LIN {X 0,Y 471.036,Z 185.812,A -85,B 0,C 180,E1 -7424.234,E2 -7424.234} C_VEL
LIN {X 0,Y 468.624,Z 186.111,A -85,B 0,C 180,E1 -7425.161,E2 -7425.161} C_VEL
LIN {X 0,Y 467.615,Z 186.239,A -85,B 0,C 180,E1 -7425.877,E2 -7425.877} C_VEL
LIN {X 0,Y 467.546,Z 186.246,A -85,B 0,C 180,E1 -7426.119,E2 -7426.119} C_VEL
LIN {X 0,Y 467.577,Z 186.237,A -85,B 0,C 180,E1 -7428.723,E2 -7428.723} C_VEL
LIN {X 0,Y 467.564,Z 186.243,A -85,B 0,C 180,E1 -7431.955,E2 -7431.955} C_VEL
LIN {X 0,Y 467.566,Z 186.241,A -85,B 0,C 180,E1 -7435.167,E2 -7435.167} C_VEL
LIN {X 0,Y 467.581,Z 186.237,A -85,B 0,C 180,E1 -7438.259,E2 -7438.259} C_VEL
LIN {X 0,Y 467.576,Z 186.241,A -85,B 0,C 180,E1 -7441.25,E2 -7441.25} C_VEL
LIN {X 0,Y 467.611,Z 186.234,A -85,B 0,C 180,E1 -7444.16,E2 -7444.16} C_VEL
LIN {X 0,Y 467.575,Z 186.24,A -85,B 0,C 180,E1 -7446.995,E2 -7446.995} C_VEL
LIN {X 0,Y 467.621,Z 186.235,A -85,B 0,C 180,E1 -7449.777,E2 -7449.777} C_VEL
LIN {X 0,Y 467.605,Z 186.234,A -85,B 0,C 180,E1 -7452.506,E2 -7452.506} C_VEL
LIN {X 0,Y 467.608,Z 186.24,A -85,B 0,C 180,E1 -7455.196,E2 -7455.196} C_VEL
LIN {X 0,Y 467.654,Z 186.229,A -85,B 0,C 180,E1 -7457.854,E2 -7457.854} C_VEL
LIN {X 0,Y 467.68,Z 186.23,A -85,B 0,C 180,E1 -7461.357,E2 -7461.357} C_VEL
LIN {X 0,Y 467.743,Z 186.217,A -85,B 0,C 180,E1 -7463.962,E2 -7463.962} C_VEL
LIN {X 0,Y 467.857,Z 186.206,A -85,B 0,C 180,E1 -7467.417,E2 -7467.417} C_VEL
LIN {X 0,Y 467.88,Z 186.199,A -85,B 0,C 180,E1 -7469.999,E2 -7469.999} C_VEL
LIN {X 0,Y 467.857,Z 186.204,A -85,B 0,C 180,E1 -7472.582,E2 -7472.582} C_VEL
LIN {X 0,Y 467.732,Z 186.218,A -85,B 0,C 180,E1 -7476.037,E2 -7476.037} C_VEL
LIN {X 0,Y 467.678,Z 186.228,A -85,B 0,C 180,E1 -7478.642,E2 -7478.642} C_VEL
LIN {X 0,Y 467.652,Z 186.228,A -85,B 0,C 180,E1 -7482.145,E2 -7482.145} C_VEL
LIN {X 0,Y 467.635,Z 186.23,A -85,B 0,C 180,E1 -7485.694,E2 -7485.694} C_VEL
LIN {X 0,Y 467.613,Z 186.241,A -85,B 0,C 180,E1 -7488.764,E2 -7488.764} C_VEL
LIN {X 0,Y 467.576,Z 186.239,A -85,B 0,C 180,E1 -7491.268,E2 -7491.268} C_VEL
LIN {X 0,Y 467.568,Z 186.238,A -85,B 0,C 180,E1 -7493.943,E2 -7493.943} C_VEL
LIN {X 0,Y 467.623,Z 186.238,A -85,B 0,C 180,E1 -7496.799,E2 -7496.799} C_VEL
LIN {X 0,Y 467.548,Z 186.241,A -85,B 0,C 180,E1 -7499.737,E2 -7499.737} C_VEL
LIN {X 0,Y 467.577,Z 186.243,A -85,B 0,C 180,E1 -7502.758,E2 -7502.758} C_VEL
LIN {X 0,Y 467.55,Z 186.241,A -85,B 0,C 180,E1 -7505.889,E2 -7505.889} C_VEL
LIN {X 0,Y 467.592,Z 186.236,A -85,B 0,C 180,E1 -7509.142,E2 -7509.142} C_VEL
LIN {X 0,Y 467.611,Z 186.239,A -85,B 0,C 180,E1 -7512.571,E2 -7512.571} C_VEL
LIN {X 0,Y 467.562,Z 186.24,A -85,B 0,C 180,E1 -7515.053,E2 -7515.053} C_VEL
LIN {X 0,Y 467.58,Z 186.237,A -85,B 0,C 180,E1 -7517.44,E2 -7517.44} C_VEL
LIN {X 0,Y 467.591,Z 186.237,A -85,B 0,C 180,E1 -7520.857,E2 -7520.857} C_VEL
LIN {X 0,Y 467.555,Z 186.248,A -85,B 0,C 180,E1 -7524.26,E2 -7524.26} C_VEL
LIN {X 0,Y 467.574,Z 186.237,A -85,B 0,C 180,E1 -7527.321,E2 -7527.321} C_VEL
LIN {X 0,Y 467.569,Z 186.24,A -85,B 0,C 180,E1 -7530.665,E2 -7530.665} C_VEL
LIN {X 0,Y 467.607,Z 186.233,A -85,B 0,C 180,E1 -7533.2,E2 -7533.2} C_VEL
LIN {X 0,Y 467.584,Z 186.239,A -85,B 0,C 180,E1 -7536.468,E2 -7536.468} C_VEL
LIN {X 0,Y 467.615,Z 186.237,A -85,B 0,C 180,E1 -7539.777,E2 -7539.777} C_VEL
LIN {X 0,Y 467.6,Z 186.236,A -85,B 0,C 180,E1 -7542.507,E2 -7542.507} C_VEL
LIN {X 0,Y 467.597,Z 186.235,A -85,B 0,C 180,E1 -7545.197,E2 -7545.197} C_VEL
LIN {X 0,Y 467.648,Z 186.236,A -85,B 0,C 180,E1 -7547.855,E2 -7547.855} C_VEL
LIN {X 0,Y 467.673,Z 186.227,A -85,B 0,C 180,E1 -7551.358,E2 -7551.358} C_VEL
LIN {X 0,Y 467.734,Z 186.223,A -85,B 0,C 180,E1 -7553.963,E2 -7553.963} C_VEL
LIN {X 0,Y 467.85,Z 186.207,A -85,B 0,C 180,E1 -7557.417,E2 -7557.417} C_VEL
LIN {X 0,Y 467.873,Z 186.204,A -85,B 0,C 180,E1 -7560,E2 -7560} C_VEL
LIN {X 0,Y 467.851,Z 186.203,A -85,B 0,C 180,E1 -7562.583,E2 -7562.583} C_VEL
LIN {X 0,Y 467.726,Z 186.221,A -85,B 0,C 180,E1 -7566.038,E2 -7566.038} C_VEL
LIN {X 0,Y 467.672,Z 186.225,A -85,B 0,C 180,E1 -7568.643,E2 -7568.643} C_VEL
LIN {X 0,Y 467.648,Z 186.229,A -85,B 0,C 180,E1 -7572.146,E2 -7572.146} C_VEL
LIN {X 0,Y 467.631,Z 186.235,A -85,B 0,C 180,E1 -7575.696,E2 -7575.696} C_VEL
LIN {X 0,Y 467.61,Z 186.234,A -85,B 0,C 180,E1 -7578.765,E2 -7578.765} C_VEL
LIN {X 0,Y 467.573,Z 186.245,A -85,B 0,C 180,E1 -7581.269,E2 -7581.269} C_VEL
LIN {X 0,Y 467.563,Z 186.24,A -85,B 0,C 180,E1 -7583.944,E2 -7583.944} C_VEL
LIN {X 0,Y 467.609,Z 186.235,A -85,B 0,C 180,E1 -7586.801,E2 -7586.801} C_VEL
LIN {X 0,Y 467.547,Z 186.242,A -85,B 0,C 180,E1 -7589.739,E2 -7589.739} C_VEL
LIN {X 0,Y 467.573,Z 186.24,A -85,B 0,C 180,E1 -7592.76,E2 -7592.76} C_VEL
LIN {X 0,Y 467.547,Z 186.241,A -85,B 0,C 180,E1 -7595.891,E2 -7595.891} C_VEL
LIN {X 0,Y 467.571,Z 186.245,A -85,B 0,C 180,E1 -7599.146,E2 -7599.146} C_VEL
LIN {X 0,Y 467.583,Z 186.239,A -85,B 0,C 180,E1 -7602.568,E2 -7602.568} C_VEL
LIN {X 0,Y 467.567,Z 186.245,A -85,B 0,C 180,E1 -7605.054,E2 -7605.054} C_VEL
LIN {X 0,Y 467.569,Z 186.242,A -85,B 0,C 180,E1 -7608.598,E2 -7608.598} C_VEL
LIN {X 0,Y 467.559,Z 186.239,A -85,B 0,C 180,E1 -7611.956,E2 -7611.956} C_VEL
LIN {X 0,Y 467.561,Z 186.245,A -85,B 0,C 180,E1 -7615.168,E2 -7615.168} C_VEL
LIN {X 0,Y 467.581,Z 186.242,A -85,B 0,C 180,E1 -7618.261,E2 -7618.261} C_VEL
LIN {X 0,Y 467.555,Z 186.247,A -85,B 0,C 180,E1 -7621.25,E2 -7621.25} C_VEL
LIN {X 0,Y 467.616,Z 186.484,A -85,B 0,C 180,E1 -7622.478,E2 -7622.478} C_VEL
LIN {X 0,Y 471.107,Z 202.041,A -85,B 0,C 180,E1 -7624.84,E2 -7624.84} C_VEL
LIN {X 0,Y 470.606,Z 215.622,A -85,B 0,C 180,E1 -7626.688,E2 -7626.688} C_VEL
LIN {X 0,Y 469.516,Z 239.357,A -85,B 0,C 180,E1 -7629.863,E2 -7629.863} C_VEL
LIN {X 0,Y 468.66,Z 261.512,A -85,B 0,C 180,E1 -7632.796,E2 -7632.796} C_VEL
LIN {X 0,Y 468.555,Z 265.454,A -85,B 0,C 180,E1 -7633.297,E2 -7633.297} C_VEL
LIN {X 0,Y 470.521,Z 284.051,A -85,B 0,C 180,E1 -7633.671,E2 -7633.671} C_VEL
LIN {X 0,Y 469.828,Z 373.176,A -85,B 0,C 180,E1 -7635.103,E2 -7635.103} C_VEL
LIN {X 0,Y 469.492,Z 386.416,A -85,B 0,C 180,E1 -7635.48,E2 -7635.48} C_VEL
LIN {X 0,Y 469.075,Z 399.132,A -85,B 0,C 180,E1 -7636.02,E2 -7636.02} C_VEL
LIN {X 0,Y 468.644,Z 410.397,A -85,B 0,C 180,E1 -7636.67,E2 -7636.67} C_VEL
LIN {X 0,Y 468.245,Z 421.339,A -85,B 0,C 180,E1 -7637.479,E2 -7637.479} C_VEL
LIN {X 0,Y 467.741,Z 432.571,A -85,B 0,C 180,E1 -7638.517,E2 -7638.517} C_VEL
LIN {X 0,Y 467.393,Z 441.968,A -85,B 0,C 180,E1 -7639.605,E2 -7639.605} C_VEL
LIN {X 0,Y 467.101,Z 451.067,A -85,B 0,C 180,E1 -7640.911,E2 -7640.911} C_VEL
LIN {X 0,Y 466.93,Z 458.368,A -85,B 0,C 180,E1 -7642.215,E2 -7642.215} C_VEL
LIN {X 0,Y 466.842,Z 464.127,A -85,B 0,C 180,E1 -7643.51,E2 -7643.51} C_VEL
LIN {X 0,Y 466.787,Z 468.686,A -85,B 0,C 180,E1 -7644.818,E2 -7644.818} C_VEL
LIN {X 0,Y 466.785,Z 471.065,A -85,B 0,C 180,E1 -7645.683,E2 -7645.683} C_VEL
LIN {X 0,Y 466.872,Z 473.007,A -85,B 0,C 180,E1 -7646.549,E2 -7646.549} C_VEL
LIN {X 0,Y 466.84,Z 474.474,A -85,B 0,C 180,E1 -7647.412,E2 -7647.412} C_VEL
LIN {X 0,Y 466.727,Z 476.099,A -85,B 0,C 180,E1 -7649.138,E2 -7649.138} C_VEL
LIN {X 0,Y 466.746,Z 476.31,A -85,B 0,C 180,E1 -7650.001,E2 -7650.001} C_VEL
LIN {X 0,Y 466.73,Z 476.064,A -85,B 0,C 180,E1 -7650.863,E2 -7650.863} C_VEL
LIN {X 0,Y 466.843,Z 474.348,A -85,B 0,C 180,E1 -7652.589,E2 -7652.589} C_VEL
LIN {X 0,Y 466.886,Z 472.858,A -85,B 0,C 180,E1 -7653.453,E2 -7653.453} C_VEL
LIN {X 0,Y 466.748,Z 469.736,A -85,B 0,C 180,E1 -7654.751,E2 -7654.751} C_VEL
LIN {X 0,Y 466.788,Z 465.534,A -85,B 0,C 180,E1 -7656.05,E2 -7656.05} C_VEL
LIN {X 0,Y 466.931,Z 460.123,A -85,B 0,C 180,E1 -7657.351,E2 -7657.351} C_VEL
LIN {X 0,Y 467.007,Z 453.309,A -85,B 0,C 180,E1 -7658.656,E2 -7658.656} C_VEL
LIN {X 0,Y 467.237,Z 444.849,A -85,B 0,C 180,E1 -7659.962,E2 -7659.962} C_VEL
LIN {X 0,Y 467.616,Z 436.186,A -85,B 0,C 180,E1 -7661.048,E2 -7661.048} C_VEL
LIN {X 0,Y 467.936,Z 427.836,A -85,B 0,C 180,E1 -7661.919,E2 -7661.919} C_VEL
LIN {X 0,Y 468.328,Z 416.572,A -85,B 0,C 180,E1 -7662.876,E2 -7662.876} C_VEL
LIN {X 0,Y 468.788,Z 404.931,A -85,B 0,C 180,E1 -7663.658,E2 -7663.658} C_VEL
LIN {X 0,Y 469.334,Z 392.149,A -85,B 0,C 180,E1 -7664.305,E2 -7664.305} C_VEL
LIN {X 0,Y 469.711,Z 379.318,A -85,B 0,C 180,E1 -7664.764,E2 -7664.764} C_VEL
LIN {X 0,Y 469.972,Z 365.957,A -85,B 0,C 180,E1 -7665.06,E2 -7665.06} C_VEL
LIN {X 0,Y 470.591,Z 282.438,A -85,B 0,C 180,E1 -7666.414,E2 -7666.414} C_VEL
LIN {X 0,Y 468.55,Z 264.229,A -85,B 0,C 180,E1 -7666.822,E2 -7666.822} C_VEL
LIN {X 0,Y 469.271,Z 242.062,A -85,B 0,C 180,E1 -7669.647,E2 -7669.647} C_VEL
LIN {X 0,Y 470.196,Z 217.219,A -85,B 0,C 180,E1 -7672.869,E2 -7672.869} C_VEL
LIN {X 0,Y 470.821,Z 201.375,A -85,B 0,C 180,E1 -7674.942,E2 -7674.942} C_VEL
LIN {X 0,Y 468.587,Z 190.486,A -85,B 0,C 180,E1 -7676.531,E2 -7676.531} C_VEL
LIN {X 0,Y 467.615,Z 186.372,A -85,B 0,C 180,E1 -7677.184,E2 -7677.184} C_VEL
LIN {X 0,Y 467.569,Z 186.245,A -85,B 0,C 180,E1 -7680.734,E2 -7680.734} C_VEL
LIN {X 0,Y 467.573,Z 186.243,A -85,B 0,C 180,E1 -7683.79,E2 -7683.79} C_VEL
LIN {X 0,Y 467.527,Z 186.25,A -85,B 0,C 180,E1 -7686.963,E2 -7686.963} C_VEL
LIN {X 0,Y 467.567,Z 186.241,A -85,B 0,C 180,E1 -7689.952,E2 -7689.952} C_VEL
LIN {X 0,Y 467.545,Z 186.246,A -85,B 0,C 180,E1 -7692.565,E2 -7692.565} C_VEL
LIN {X 0,Y 467.568,Z 186.246,A -85,B 0,C 180,E1 -7695.052,E2 -7695.052} C_VEL
LIN {X 0,Y 467.575,Z 186.241,A -85,B 0,C 180,E1 -7698.596,E2 -7698.596} C_VEL
LIN {X 0,Y 467.567,Z 186.239,A -85,B 0,C 180,E1 -7701.955,E2 -7701.955} C_VEL
LIN {X 0,Y 467.561,Z 186.244,A -85,B 0,C 180,E1 -7705.167,E2 -7705.167} C_VEL
LIN {X 0,Y 467.584,Z 186.24,A -85,B 0,C 180,E1 -7708.26,E2 -7708.26} C_VEL
LIN {X 0,Y 467.577,Z 186.241,A -85,B 0,C 180,E1 -7711.25,E2 -7711.25} C_VEL
LIN {X 0,Y 467.599,Z 186.238,A -85,B 0,C 180,E1 -7714.159,E2 -7714.159} C_VEL
LIN {X 0,Y 467.578,Z 186.241,A -85,B 0,C 180,E1 -7716.995,E2 -7716.995} C_VEL
LIN {X 0,Y 467.623,Z 186.233,A -85,B 0,C 180,E1 -7719.777,E2 -7719.777} C_VEL
LIN {X 0,Y 467.597,Z 186.241,A -85,B 0,C 180,E1 -7722.506,E2 -7722.506} C_VEL
LIN {X 0,Y 467.606,Z 186.237,A -85,B 0,C 180,E1 -7725.196,E2 -7725.196} C_VEL
LIN {X 0,Y 467.657,Z 186.23,A -85,B 0,C 180,E1 -7727.854,E2 -7727.854} C_VEL
LIN {X 0,Y 467.671,Z 186.228,A -85,B 0,C 180,E1 -7731.357,E2 -7731.357} C_VEL
LIN {X 0,Y 467.721,Z 186.226,A -85,B 0,C 180,E1 -7733.962,E2 -7733.962} C_VEL
LIN {X 0,Y 467.859,Z 186.208,A -85,B 0,C 180,E1 -7737.417,E2 -7737.417} C_VEL
LIN {X 0,Y 467.821,Z 186.447,A -85,B 0,C 180,E1 -7739.112,E2 -7739.112} C_VEL
LIN {X 0,Y 468.474,Z 190.11,A -85,B 0,C 180,E1 -7739.785,E2 -7739.785} C_VEL
LIN {X 0,Y 468.367,Z 206.386,A -85,B 0,C 180,E1 -7742.58,E2 -7742.58} C_VEL
LIN {X 0,Y 468.286,Z 223.54,A -85,B 0,C 180,E1 -7745.598,E2 -7745.598} C_VEL
LIN {X 0,Y 468.274,Z 227.237,A -85,B 0,C 180,E1 -7746.219,E2 -7746.219} C_VEL
LIN {X 0,Y 470.377,Z 238.502,A -85,B 0,C 180,E1 -7746.541,E2 -7746.541} C_VEL
LIN {X 0,Y 469.573,Z 308.823,A -85,B 0,C 180,E1 -7747.834,E2 -7747.834} C_VEL
LIN {X 0,Y 469.438,Z 320.442,A -85,B 0,C 180,E1 -7748.211,E2 -7748.211} C_VEL
LIN {X 0,Y 469.166,Z 332.332,A -85,B 0,C 180,E1 -7748.791,E2 -7748.791} C_VEL
LIN {X 0,Y 468.847,Z 342.842,A -85,B 0,C 180,E1 -7749.49,E2 -7749.49} C_VEL
LIN {X 0,Y 468.516,Z 353.004,A -85,B 0,C 180,E1 -7750.37,E2 -7750.37} C_VEL
LIN {X 0,Y 468.196,Z 361.041,A -85,B 0,C 180,E1 -7751.252,E2 -7751.252} C_VEL
LIN {X 0,Y 467.882,Z 368.755,A -85,B 0,C 180,E1 -7752.303,E2 -7752.303} C_VEL
LIN {X 0,Y 467.622,Z 375.472,A -85,B 0,C 180,E1 -7753.471,E2 -7753.471} C_VEL
LIN {X 0,Y 467.334,Z 381.402,A -85,B 0,C 180,E1 -7754.812,E2 -7754.812} C_VEL
LIN {X 0,Y 467.168,Z 385.738,A -85,B 0,C 180,E1 -7756.159,E2 -7756.159} C_VEL
LIN {X 0,Y 466.985,Z 388.645,A -85,B 0,C 180,E1 -7757.517,E2 -7757.517} C_VEL
LIN {X 0,Y 466.938,Z 389.95,A -85,B 0,C 180,E1 -7758.517,E2 -7758.517} C_VEL
LIN {X 0,Y 466.891,Z 390.505,A -85,B 0,C 180,E1 -7759.339,E2 -7759.339} C_VEL
LIN {X 0,Y 466.89,Z 390.575,A -85,B 0,C 180,E1 -7760.255,E2 -7760.255} C_VEL
LIN {X 0,Y 466.896,Z 390.092,A -85,B 0,C 180,E1 -7761.177,E2 -7761.177} C_VEL
LIN {X 0,Y 466.919,Z 388.996,A -85,B 0,C 180,E1 -7762.104,E2 -7762.104} C_VEL
LIN {X 0,Y 467.041,Z 386.528,A -85,B 0,C 180,E1 -7763.376,E2 -7763.376} C_VEL
LIN {X 0,Y 467.169,Z 383.529,A -85,B 0,C 180,E1 -7764.437,E2 -7764.437} C_VEL
LIN {X 0,Y 467.36,Z 378.061,A -85,B 0,C 180,E1 -7765.854,E2 -7765.854} C_VEL
LIN {X 0,Y 467.522,Z 372.051,A -85,B 0,C 180,E1 -7767.026,E2 -7767.026} C_VEL
LIN {X 0,Y 467.789,Z 365.797,A -85,B 0,C 180,E1 -7768.001,E2 -7768.001} C_VEL
LIN {X 0,Y 468.081,Z 357.37,A -85,B 0,C 180,E1 -7769.057,E2 -7769.057} C_VEL
LIN {X 0,Y 468.372,Z 348.64,A -85,B 0,C 180,E1 -7769.928,E2 -7769.928} C_VEL
LIN {X 0,Y 468.723,Z 338.054,A -85,B 0,C 180,E1 -7770.754,E2 -7770.754} C_VEL
LIN {X 0,Y 468.99,Z 327.029,A -85,B 0,C 180,E1 -7771.405,E2 -7771.405} C_VEL
LIN {X 0,Y 469.178,Z 314.743,A -85,B 0,C 180,E1 -7771.919,E2 -7771.919} C_VEL
LIN {X 0,Y 469.307,Z 301.965,A -85,B 0,C 180,E1 -7772.241,E2 -7772.241} C_VEL
LIN {X 0,Y 469.804,Z 237.356,A -85,B 0,C 180,E1 -7773.338,E2 -7773.338} C_VEL
LIN {X 0,Y 467.979,Z 226.462,A -85,B 0,C 180,E1 -7773.612,E2 -7773.612} C_VEL
LIN {X 0,Y 468.255,Z 209.645,A -85,B 0,C 180,E1 -7776.895,E2 -7776.895} C_VEL
LIN {X 0,Y 468.539,Z 193.341,A -85,B 0,C 180,E1 -7780.164,E2 -7780.164} C_VEL
LIN {X 0,Y 468.184,Z 189.189,A -85,B 0,C 180,E1 -7781.023,E2 -7781.023} C_VEL
LIN {X 0,Y 467.629,Z 186.277,A -85,B 0,C 180,E1 -7781.702,E2 -7781.702} C_VEL
LIN {X 0,Y 467.564,Z 186.243,A -85,B 0,C 180,E1 -7785.052,E2 -7785.052} C_VEL
LIN {X 0,Y 467.546,Z 186.246,A -85,B 0,C 180,E1 -7786.119,E2 -7786.119} C_VEL
LIN {X 0,Y 466.92,Z 186.33,A -85,B 0,C 180,E1 -7786.838,E2 -7786.838} C_VEL
LIN {X 0,Y 464.09,Z 186.689,A -85,B 0,C 180,E1 -7788.007,E2 -7788.007} C_VEL
LIN {X 0,Y 461.667,Z 186.988,A -85,B 0,C 180,E1 -7788.949,E2 -7788.949} C_VEL
LIN {X 0,Y 460.617,Z 187.112,A -85,B 0,C 180,E1 -7789.677,E2 -7789.677} C_VEL
LIN {X 0,Y 460.528,Z 187.12,A -85,B 0,C 180,E1 -7789.924,E2 -7789.924} C_VEL
LIN {X 0,Y 460.499,Z 187.119,A -85,B 0,C 180,E1 -7792.523,E2 -7792.523} C_VEL
LIN {X 0,Y 460.547,Z 187.121,A -85,B 0,C 180,E1 -7795.623,E2 -7795.623} C_VEL
LIN {X 0,Y 460.535,Z 187.114,A -85,B 0,C 180,E1 -7798.744,E2 -7798.744} C_VEL
LIN {X 0,Y 460.587,Z 187.108,A -85,B 0,C 180,E1 -7802.252,E2 -7802.252} C_VEL
LIN {X 0,Y 460.558,Z 187.112,A -85,B 0,C 180,E1 -7804.705,E2 -7804.705} C_VEL
LIN {X 0,Y 460.509,Z 187.124,A -85,B 0,C 180,E1 -7807.571,E2 -7807.571} C_VEL
LIN {X 0,Y 460.567,Z 187.11,A -85,B 0,C 180,E1 -7810.384,E2 -7810.384} C_VEL
LIN {X 0,Y 460.562,Z 187.116,A -85,B 0,C 180,E1 -7813.146,E2 -7813.146} C_VEL
LIN {X 0,Y 460.556,Z 187.113,A -85,B 0,C 180,E1 -7815.867,E2 -7815.867} C_VEL
LIN {X 0,Y 460.61,Z 187.106,A -85,B 0,C 180,E1 -7818.559,E2 -7818.559} C_VEL
LIN {X 0,Y 460.693,Z 187.094,A -85,B 0,C 180,E1 -7822.108,E2 -7822.108} C_VEL
LIN {X 0,Y 460.697,Z 187.097,A -85,B 0,C 180,E1 -7824.748,E2 -7824.748} C_VEL
LIN {X 0,Y 460.822,Z 187.083,A -85,B 0,C 180,E1 -7827.377,E2 -7827.377} C_VEL
LIN {X 0,Y 460.851,Z 187.075,A -85,B 0,C 180,E1 -7829.999,E2 -7829.999} C_VEL
LIN {X 0,Y 460.822,Z 187.081,A -85,B 0,C 180,E1 -7832.622,E2 -7832.622} C_VEL
LIN {X 0,Y 460.699,Z 187.094,A -85,B 0,C 180,E1 -7836.129,E2 -7836.129} C_VEL
LIN {X 0,Y 460.625,Z 187.109,A -85,B 0,C 180,E1 -7838.775,E2 -7838.775} C_VEL
LIN {X 0,Y 460.609,Z 187.108,A -85,B 0,C 180,E1 -7842.444,E2 -7842.444} C_VEL
LIN {X 0,Y 460.596,Z 187.107,A -85,B 0,C 180,E1 -7845.997,E2 -7845.997} C_VEL
LIN {X 0,Y 460.567,Z 187.117,A -85,B 0,C 180,E1 -7848.901,E2 -7848.901} C_VEL
LIN {X 0,Y 460.511,Z 187.118,A -85,B 0,C 180,E1 -7851.485,E2 -7851.485} C_VEL
LIN {X 0,Y 460.537,Z 187.117,A -85,B 0,C 180,E1 -7854.332,E2 -7854.332} C_VEL
LIN {X 0,Y 460.578,Z 187.11,A -85,B 0,C 180,E1 -7857.242,E2 -7857.242} C_VEL
LIN {X 0,Y 460.505,Z 187.121,A -85,B 0,C 180,E1 -7860.239,E2 -7860.239} C_VEL
LIN {X 0,Y 460.523,Z 187.116,A -85,B 0,C 180,E1 -7863.324,E2 -7863.324} C_VEL
LIN {X 0,Y 460.494,Z 187.121,A -85,B 0,C 180,E1 -7866.014,E2 -7866.014} C_VEL
LIN {X 0,Y 460.551,Z 187.115,A -85,B 0,C 180,E1 -7868.899,E2 -7868.899} C_VEL
LIN {X 0,Y 460.54,Z 187.118,A -85,B 0,C 180,E1 -7872.178,E2 -7872.178} C_VEL
LIN {X 0,Y 460.509,Z 187.117,A -85,B 0,C 180,E1 -7875.411,E2 -7875.411} C_VEL
LIN {X 0,Y 460.527,Z 187.122,A -85,B 0,C 180,E1 -7878.397,E2 -7878.397} C_VEL
LIN {X 0,Y 460.531,Z 187.115,A -85,B 0,C 180,E1 -7881.268,E2 -7881.268} C_VEL
LIN {X 0,Y 460.505,Z 187.122,A -85,B 0,C 180,E1 -7884.554,E2 -7884.554} C_VEL
LIN {X 0,Y 460.524,Z 187.118,A -85,B 0,C 180,E1 -7887.716,E2 -7887.716} C_VEL
LIN {X 0,Y 460.538,Z 187.115,A -85,B 0,C 180,E1 -7890.769,E2 -7890.769} C_VEL
LIN {X 0,Y 460.554,Z 187.115,A -85,B 0,C 180,E1 -7893.735,E2 -7893.735} C_VEL
LIN {X 0,Y 460.537,Z 187.115,A -85,B 0,C 180,E1 -7896.624,E2 -7896.624} C_VEL
LIN {X 0,Y 460.543,Z 187.115,A -85,B 0,C 180,E1 -7899.453,E2 -7899.453} C_VEL
LIN {X 0,Y 460.551,Z 187.117,A -85,B 0,C 180,E1 -7902.23,E2 -7902.23} C_VEL
LIN {X 0,Y 460.56,Z 187.111,A -85,B 0,C 180,E1 -7904.965,E2 -7904.965} C_VEL
LIN {X 0,Y 460.605,Z 187.106,A -85,B 0,C 180,E1 -7908.56,E2 -7908.56} C_VEL
LIN {X 0,Y 460.686,Z 187.099,A -85,B 0,C 180,E1 -7912.109,E2 -7912.109} C_VEL
LIN {X 0,Y 460.688,Z 187.095,A -85,B 0,C 180,E1 -7914.749,E2 -7914.749} C_VEL
LIN {X 0,Y 460.791,Z 187.086,A -85,B 0,C 180,E1 -7917.378,E2 -7917.378} C_VEL
LIN {X 0,Y 460.844,Z 187.079,A -85,B 0,C 180,E1 -7920,E2 -7920} C_VEL
LIN {X 0,Y 460.792,Z 187.082,A -85,B 0,C 180,E1 -7922.623,E2 -7922.623} C_VEL
LIN {X 0,Y 460.693,Z 187.096,A -85,B 0,C 180,E1 -7926.131,E2 -7926.131} C_VEL
LIN {X 0,Y 460.62,Z 187.104,A -85,B 0,C 180,E1 -7928.777,E2 -7928.777} C_VEL
LIN {X 0,Y 460.606,Z 187.105,A -85,B 0,C 180,E1 -7932.446,E2 -7932.446} C_VEL
LIN {X 0,Y 460.593,Z 187.108,A -85,B 0,C 180,E1 -7935.998,E2 -7935.998} C_VEL
LIN {X 0,Y 460.563,Z 187.113,A -85,B 0,C 180,E1 -7938.902,E2 -7938.902} C_VEL
LIN {X 0,Y 460.509,Z 187.124,A -85,B 0,C 180,E1 -7941.486,E2 -7941.486} C_VEL
LIN {X 0,Y 460.533,Z 187.114,A -85,B 0,C 180,E1 -7944.333,E2 -7944.333} C_VEL
LIN {X 0,Y 460.566,Z 187.119,A -85,B 0,C 180,E1 -7947.245,E2 -7947.245} C_VEL
LIN {X 0,Y 460.504,Z 187.118,A -85,B 0,C 180,E1 -7950.241,E2 -7950.241} C_VEL
LIN {X 0,Y 460.514,Z 187.123,A -85,B 0,C 180,E1 -7953.327,E2 -7953.327} C_VEL
LIN {X 0,Y 460.471,Z 187.124,A -85,B 0,C 180,E1 -7956.53,E2 -7956.53} C_VEL
LIN {X 0,Y 460.522,Z 187.116,A -85,B 0,C 180,E1 -7959.864,E2 -7959.864} C_VEL
LIN {X 0,Y 460.509,Z 187.124,A -85,B 0,C 180,E1 -7962.901,E2 -7962.901} C_VEL
LIN {X 0,Y 460.504,Z 187.118,A -85,B 0,C 180,E1 -7965.832,E2 -7965.832} C_VEL
LIN {X 0,Y 460.523,Z 187.123,A -85,B 0,C 180,E1 -7968.989,E2 -7968.989} C_VEL
LIN {X 0,Y 460.518,Z 187.119,A -85,B 0,C 180,E1 -7971.267,E2 -7971.267} C_VEL
LIN {X 0,Y 460.506,Z 187.122,A -85,B 0,C 180,E1 -7974.555,E2 -7974.555} C_VEL
LIN {X 0,Y 460.529,Z 187.118,A -85,B 0,C 180,E1 -7977.717,E2 -7977.717} C_VEL
LIN {X 0,Y 460.525,Z 187.121,A -85,B 0,C 180,E1 -7980.769,E2 -7980.769} C_VEL
LIN {X 0,Y 460.592,Z 187.302,A -85,B 0,C 180,E1 -7982.221,E2 -7982.221} C_VEL
LIN {X 0,Y 464.139,Z 203.176,A -85,B 0,C 180,E1 -7984.675,E2 -7984.675} C_VEL
LIN {X 0,Y 464.098,Z 208.615,A -85,B 0,C 180,E1 -7985.437,E2 -7985.437} C_VEL
LIN {X 0,Y 463.023,Z 230.345,A -85,B 0,C 180,E1 -7988.407,E2 -7988.407} C_VEL
LIN {X 0,Y 461.919,Z 255.678,A -85,B 0,C 180,E1 -7991.827,E2 -7991.827} C_VEL
LIN {X 0,Y 461.554,Z 265.337,A -85,B 0,C 180,E1 -7993.085,E2 -7993.085} C_VEL
LIN {X 0,Y 463.632,Z 284.318,A -85,B 0,C 180,E1 -7993.477,E2 -7993.477} C_VEL
LIN {X 0,Y 462.886,Z 373.252,A -85,B 0,C 180,E1 -7994.93,E2 -7994.93} C_VEL
LIN {X 0,Y 462.514,Z 386.288,A -85,B 0,C 180,E1 -7995.312,E2 -7995.312} C_VEL
LIN {X 0,Y 462.1,Z 398.896,A -85,B 0,C 180,E1 -7995.861,E2 -7995.861} C_VEL
LIN {X 0,Y 461.613,Z 410.875,A -85,B 0,C 180,E1 -7996.575,E2 -7996.575} C_VEL
LIN {X 0,Y 461.202,Z 421.571,A -85,B 0,C 180,E1 -7997.391,E2 -7997.391} C_VEL
LIN {X 0,Y 460.659,Z 431.622,A -85,B 0,C 180,E1 -7998.338,E2 -7998.338} C_VEL
LIN {X 0,Y 460.371,Z 441.117,A -85,B 0,C 180,E1 -7999.445,E2 -7999.445} C_VEL
LIN {X 0,Y 460.026,Z 450.256,A -85,B 0,C 180,E1 -8000.77,E2 -8000.77} C_VEL
LIN {X 0,Y 459.866,Z 457.603,A -85,B 0,C 180,E1 -8002.095,E2 -8002.095} C_VEL
LIN {X 0,Y 459.764,Z 463.797,A -85,B 0,C 180,E1 -8003.515,E2 -8003.515} C_VEL
LIN {X 0,Y 459.724,Z 467.987,A -85,B 0,C 180,E1 -8004.738,E2 -8004.738} C_VEL
LIN {X 0,Y 459.69,Z 470.374,A -85,B 0,C 180,E1 -8005.617,E2 -8005.617} C_VEL
LIN {X 0,Y 459.794,Z 472.326,A -85,B 0,C 180,E1 -8006.495,E2 -8006.495} C_VEL
LIN {X 0,Y 459.784,Z 473.81,A -85,B 0,C 180,E1 -8007.372,E2 -8007.372} C_VEL
LIN {X 0,Y 459.656,Z 475.441,A -85,B 0,C 180,E1 -8009.125,E2 -8009.125} C_VEL
LIN {X 0,Y 459.676,Z 475.656,A -85,B 0,C 180,E1 -8010.001,E2 -8010.001} C_VEL
LIN {X 0,Y 459.659,Z 475.414,A -85,B 0,C 180,E1 -8010.877,E2 -8010.877} C_VEL
LIN {X 0,Y 459.787,Z 473.699,A -85,B 0,C 180,E1 -8012.629,E2 -8012.629} C_VEL
LIN {X 0,Y 459.807,Z 472.206,A -85,B 0,C 180,E1 -8013.506,E2 -8013.506} C_VEL
LIN {X 0,Y 459.673,Z 469.078,A -85,B 0,C 180,E1 -8014.824,E2 -8014.824} C_VEL
LIN {X 0,Y 459.711,Z 464.867,A -85,B 0,C 180,E1 -8016.144,E2 -8016.144} C_VEL
LIN {X 0,Y 459.833,Z 459.444,A -85,B 0,C 180,E1 -8017.465,E2 -8017.465} C_VEL
LIN {X 0,Y 459.947,Z 452.625,A -85,B 0,C 180,E1 -8018.79,E2 -8018.79} C_VEL
LIN {X 0,Y 460.206,Z 444.16,A -85,B 0,C 180,E1 -8020.115,E2 -8020.115} C_VEL
LIN {X 0,Y 460.624,Z 434.49,A -85,B 0,C 180,E1 -8021.329,E2 -8021.329} C_VEL
LIN {X 0,Y 461.08,Z 424.743,A -85,B 0,C 180,E1 -8022.322,E2 -8022.322} C_VEL
LIN {X 0,Y 461.433,Z 414.081,A -85,B 0,C 180,E1 -8023.207,E2 -8023.207} C_VEL
LIN {X 0,Y 461.958,Z 402.301,A -85,B 0,C 180,E1 -8023.976,E2 -8023.976} C_VEL
LIN {X 0,Y 462.448,Z 390.033,A -85,B 0,C 180,E1 -8024.579,E2 -8024.579} C_VEL
LIN {X 0,Y 462.909,Z 377.557,A -85,B 0,C 180,E1 -8025.014,E2 -8025.014} C_VEL
LIN {X 0,Y 463.112,Z 364.931,A -85,B 0,C 180,E1 -8025.289,E2 -8025.289} C_VEL
LIN {X 0,Y 463.725,Z 282.766,A -85,B 0,C 180,E1 -8026.651,E2 -8026.651} C_VEL
LIN {X 0,Y 461.606,Z 263.985,A -85,B 0,C 180,E1 -8027.083,E2 -8027.083} C_VEL
LIN {X 0,Y 462.408,Z 241.394,A -85,B 0,C 180,E1 -8029.997,E2 -8029.997} C_VEL
LIN {X 0,Y 463.395,Z 216.884,A -85,B 0,C 180,E1 -8033.224,E2 -8033.224} C_VEL
LIN {X 0,Y 463.975,Z 202.863,A -85,B 0,C 180,E1 -8035.096,E2 -8035.096} C_VEL
LIN {X 0,Y 461.317,Z 190.433,A -85,B 0,C 180,E1 -8036.951,E2 -8036.951} C_VEL
LIN {X 0,Y 460.565,Z 187.243,A -85,B 0,C 180,E1 -8037.488,E2 -8037.488} C_VEL
LIN {X 0,Y 460.507,Z 187.123,A -85,B 0,C 180,E1 -8040.241,E2 -8040.241} C_VEL
LIN {X 0,Y 460.523,Z 187.123,A -85,B 0,C 180,E1 -8043.326,E2 -8043.326} C_VEL
LIN {X 0,Y 460.476,Z 187.127,A -85,B 0,C 180,E1 -8046.53,E2 -8046.53} C_VEL
LIN {X 0,Y 460.516,Z 187.12,A -85,B 0,C 180,E1 -8049.864,E2 -8049.864} C_VEL
LIN {X 0,Y 460.482,Z 187.127,A -85,B 0,C 180,E1 -8052.896,E2 -8052.896} C_VEL
LIN {X 0,Y 460.508,Z 187.119,A -85,B 0,C 180,E1 -8055.831,E2 -8055.831} C_VEL
LIN {X 0,Y 460.529,Z 187.123,A -85,B 0,C 180,E1 -8058.988,E2 -8058.988} C_VEL
LIN {X 0,Y 460.523,Z 187.12,A -85,B 0,C 180,E1 -8061.266,E2 -8061.266} C_VEL
LIN {X 0,Y 460.511,Z 187.121,A -85,B 0,C 180,E1 -8064.554,E2 -8064.554} C_VEL
LIN {X 0,Y 460.532,Z 187.116,A -85,B 0,C 180,E1 -8067.715,E2 -8067.715} C_VEL
LIN {X 0,Y 460.54,Z 187.119,A -85,B 0,C 180,E1 -8070.769,E2 -8070.769} C_VEL
LIN {X 0,Y 460.558,Z 187.113,A -85,B 0,C 180,E1 -8073.734,E2 -8073.734} C_VEL
LIN {X 0,Y 460.546,Z 187.119,A -85,B 0,C 180,E1 -8076.624,E2 -8076.624} C_VEL
LIN {X 0,Y 460.552,Z 187.114,A -85,B 0,C 180,E1 -8079.452,E2 -8079.452} C_VEL
LIN {X 0,Y 460.549,Z 187.119,A -85,B 0,C 180,E1 -8082.229,E2 -8082.229} C_VEL
LIN {X 0,Y 460.565,Z 187.116,A -85,B 0,C 180,E1 -8084.964,E2 -8084.964} C_VEL
LIN {X 0,Y 460.612,Z 187.111,A -85,B 0,C 180,E1 -8088.559,E2 -8088.559} C_VEL
LIN {X 0,Y 460.621,Z 187.107,A -85,B 0,C 180,E1 -8091.223,E2 -8091.223} C_VEL
LIN {X 0,Y 460.685,Z 187.102,A -85,B 0,C 180,E1 -8093.869,E2 -8093.869} C_VEL
LIN {X 0,Y 460.8,Z 187.088,A -85,B 0,C 180,E1 -8097.377,E2 -8097.377} C_VEL
LIN {X 0,Y 460.761,Z 187.273,A -85,B 0,C 180,E1 -8098.852,E2 -8098.852} C_VEL
LIN {X 0,Y 461.601,Z 192.233,A -85,B 0,C 180,E1 -8099.781,E2 -8099.781} C_VEL
LIN {X 0,Y 461.441,Z 208.622,A -85,B 0,C 180,E1 -8102.618,E2 -8102.618} C_VEL
LIN {X 0,Y 461.386,Z 227.376,A -85,B 0,C 180,E1 -8105.928,E2 -8105.928} C_VEL
LIN {X 0,Y 461.975,Z 230.575,A -85,B 0,C 180,E1 -8106.058,E2 -8106.058} C_VEL
LIN {X 0,Y 463.634,Z 239.773,A -85,B 0,C 180,E1 -8106.309,E2 -8106.309} C_VEL
LIN {X 0,Y 462.725,Z 309.039,A -85,B 0,C 180,E1 -8107.609,E2 -8107.609} C_VEL
LIN {X 0,Y 462.581,Z 320.813,A -85,B 0,C 180,E1 -8107.994,E2 -8107.994} C_VEL
LIN {X 0,Y 462.322,Z 331.908,A -85,B 0,C 180,E1 -8108.534,E2 -8108.534} C_VEL
LIN {X 0,Y 462.046,Z 341.968,A -85,B 0,C 180,E1 -8109.189,E2 -8109.189} C_VEL
LIN {X 0,Y 461.659,Z 352.432,A -85,B 0,C 180,E1 -8110.082,E2 -8110.082} C_VEL
LIN {X 0,Y 461.307,Z 360.719,A -85,B 0,C 180,E1 -8110.978,E2 -8110.978} C_VEL
LIN {X 0,Y 460.922,Z 368.984,A -85,B 0,C 180,E1 -8112.102,E2 -8112.102} C_VEL
LIN {X 0,Y 460.633,Z 375.506,A -85,B 0,C 180,E1 -8113.229,E2 -8113.229} C_VEL
LIN {X 0,Y 460.348,Z 381.596,A -85,B 0,C 180,E1 -8114.59,E2 -8114.59} C_VEL
LIN {X 0,Y 460.125,Z 386.051,A -85,B 0,C 180,E1 -8115.958,E2 -8115.958} C_VEL
LIN {X 0,Y 460.044,Z 388.224,A -85,B 0,C 180,E1 -8116.873,E2 -8116.873} C_VEL
LIN {X 0,Y 459.9,Z 389.833,A -85,B 0,C 180,E1 -8117.796,E2 -8117.796} C_VEL
LIN {X 0,Y 459.873,Z 390.817,A -85,B 0,C 180,E1 -8118.719,E2 -8118.719} C_VEL
LIN {X 0,Y 459.822,Z 391.255,A -85,B 0,C 180,E1 -8119.648,E2 -8119.648} C_VEL
LIN {X 0,Y 459.828,Z 391.134,A -85,B 0,C 180,E1 -8120.581,E2 -8120.581} C_VEL
LIN {X 0,Y 459.847,Z 390.402,A -85,B 0,C 180,E1 -8121.518,E2 -8121.518} C_VEL
LIN {X 0,Y 459.892,Z 389.094,A -85,B 0,C 180,E1 -8122.46,E2 -8122.46} C_VEL
LIN {X 0,Y 460.06,Z 385.889,A -85,B 0,C 180,E1 -8123.906,E2 -8123.906} C_VEL
LIN {X 0,Y 460.215,Z 381.211,A -85,B 0,C 180,E1 -8125.314,E2 -8125.314} C_VEL
LIN {X 0,Y 460.385,Z 375.853,A -85,B 0,C 180,E1 -8126.52,E2 -8126.52} C_VEL
LIN {X 0,Y 460.683,Z 368.656,A -85,B 0,C 180,E1 -8127.77,E2 -8127.77} C_VEL
LIN {X 0,Y 460.998,Z 359.912,A -85,B 0,C 180,E1 -8128.949,E2 -8128.949} C_VEL
LIN {X 0,Y 461.337,Z 350.946,A -85,B 0,C 180,E1 -8129.9,E2 -8129.9} C_VEL
LIN {X 0,Y 461.716,Z 340.258,A -85,B 0,C 180,E1 -8130.785,E2 -8130.785} C_VEL
LIN {X 0,Y 461.99,Z 328.755,A -85,B 0,C 180,E1 -8131.501,E2 -8131.501} C_VEL
LIN {X 0,Y 462.235,Z 316.882,A -85,B 0,C 180,E1 -8132.025,E2 -8132.025} C_VEL
LIN {X 0,Y 462.353,Z 304.825,A -85,B 0,C 180,E1 -8132.367,E2 -8132.367} C_VEL
LIN {X 0,Y 462.925,Z 238.264,A -85,B 0,C 180,E1 -8133.525,E2 -8133.525} C_VEL
LIN {X 0,Y 460.989,Z 226.979,A -85,B 0,C 180,E1 -8133.806,E2 -8133.806} C_VEL
LIN {X 0,Y 460.961,Z 225.683,A -85,B 0,C 180,E1 -8133.985,E2 -8133.985} C_VEL
LIN {X 0,Y 461.343,Z 207.814,A -85,B 0,C 180,E1 -8137.542,E2 -8137.542} C_VEL
LIN {X 0,Y 461.532,Z 192.652,A -85,B 0,C 180,E1 -8140.617,E2 -8140.617} C_VEL
LIN {X 0,Y 460.59,Z 187.186,A -85,B 0,C 180,E1 -8141.837,E2 -8141.837} C_VEL
LIN {X 0,Y 460.512,Z 187.123,A -85,B 0,C 180,E1 -8145.411,E2 -8145.411} C_VEL
LIN {X 0,Y 460.53,Z 187.116,A -85,B 0,C 180,E1 -8148.397,E2 -8148.397} C_VEL
LIN {X 0,Y 460.528,Z 187.12,A -85,B 0,C 180,E1 -8149.924,E2 -8149.924} C_VEL
LIN {X 0,Y 459.847,Z 187.201,A -85,B 0,C 180,E1 -8150.654,E2 -8150.654} C_VEL
LIN {X 0,Y 456.979,Z 187.564,A -85,B 0,C 180,E1 -8151.839,E2 -8151.839} C_VEL
LIN {X 0,Y 454.564,Z 187.87,A -85,B 0,C 180,E1 -8152.795,E2 -8152.795} C_VEL
LIN {X 0,Y 453.534,Z 187.995,A -85,B 0,C 180,E1 -8153.534,E2 -8153.534} C_VEL
LIN {X 0,Y 453.453,Z 188.003,A -85,B 0,C 180,E1 -8153.784,E2 -8153.784} C_VEL
LIN {X 0,Y 453.489,Z 187.992,A -85,B 0,C 180,E1 -8156.81,E2 -8156.81} C_VEL
LIN {X 0,Y 453.473,Z 187.994,A -85,B 0,C 180,E1 -8160.268,E2 -8160.268} C_VEL
LIN {X 0,Y 453.513,Z 187.994,A -85,B 0,C 180,E1 -8163.294,E2 -8163.294} C_VEL
LIN {X 0,Y 453.501,Z 187.991,A -85,B 0,C 180,E1 -8166.238,E2 -8166.238} C_VEL
LIN {X 0,Y 453.481,Z 187.997,A -85,B 0,C 180,E1 -8169.117,E2 -8169.117} C_VEL
LIN {X 0,Y 453.509,Z 187.991,A -85,B 0,C 180,E1 -8171.944,E2 -8171.944} C_VEL
LIN {X 0,Y 453.54,Z 187.987,A -85,B 0,C 180,E1 -8174.726,E2 -8174.726} C_VEL
LIN {X 0,Y 453.558,Z 187.983,A -85,B 0,C 180,E1 -8178.378,E2 -8178.378} C_VEL
LIN {X 0,Y 453.65,Z 187.972,A -85,B 0,C 180,E1 -8181.985,E2 -8181.985} C_VEL
LIN {X 0,Y 453.67,Z 187.971,A -85,B 0,C 180,E1 -8184.666,E2 -8184.666} C_VEL
LIN {X 0,Y 453.762,Z 187.963,A -85,B 0,C 180,E1 -8187.336,E2 -8187.336} C_VEL
LIN {X 0,Y 453.821,Z 187.951,A -85,B 0,C 180,E1 -8189.999,E2 -8189.999} C_VEL
LIN {X 0,Y 453.763,Z 187.961,A -85,B 0,C 180,E1 -8192.663,E2 -8192.663} C_VEL
LIN {X 0,Y 453.666,Z 187.97,A -85,B 0,C 180,E1 -8196.225,E2 -8196.225} C_VEL
LIN {X 0,Y 453.589,Z 187.987,A -85,B 0,C 180,E1 -8198.913,E2 -8198.913} C_VEL
LIN {X 0,Y 453.559,Z 187.987,A -85,B 0,C 180,E1 -8202.528,E2 -8202.528} C_VEL
LIN {X 0,Y 453.54,Z 187.987,A -85,B 0,C 180,E1 -8206.195,E2 -8206.195} C_VEL
LIN {X 0,Y 453.516,Z 187.993,A -85,B 0,C 180,E1 -8209.04,E2 -8209.04} C_VEL
LIN {X 0,Y 453.471,Z 187.994,A -85,B 0,C 180,E1 -8211.835,E2 -8211.835} C_VEL
LIN {X 0,Y 453.509,Z 187.997,A -85,B 0,C 180,E1 -8214.734,E2 -8214.734} C_VEL
LIN {X 0,Y 453.532,Z 187.987,A -85,B 0,C 180,E1 -8217.96,E2 -8217.96} C_VEL
LIN {X 0,Y 453.46,Z 187.995,A -85,B 0,C 180,E1 -8221.525,E2 -8221.525} C_VEL
LIN {X 0,Y 453.496,Z 187.996,A -85,B 0,C 180,E1 -8224.78,E2 -8224.78} C_VEL
LIN {X 0,Y 453.474,Z 187.999,A -85,B 0,C 180,E1 -8228.309,E2 -8228.309} C_VEL
LIN {X 0,Y 453.509,Z 187.995,A -85,B 0,C 180,E1 -8230.606,E2 -8230.606} C_VEL
LIN {X 0,Y 453.474,Z 187.994,A -85,B 0,C 180,E1 -8233.247,E2 -8233.247} C_VEL
LIN {X 0,Y 453.458,Z 187.997,A -85,B 0,C 180,E1 -8235.779,E2 -8235.779} C_VEL
LIN {X 0,Y 453.508,Z 187.99,A -85,B 0,C 180,E1 -8239.405,E2 -8239.405} C_VEL
LIN {X 0,Y 453.468,Z 188.002,A -85,B 0,C 180,E1 -8242.223,E2 -8242.223} C_VEL
LIN {X 0,Y 453.481,Z 187.993,A -85,B 0,C 180,E1 -8245.222,E2 -8245.222} C_VEL
LIN {X 0,Y 453.476,Z 187.998,A -85,B 0,C 180,E1 -8248.471,E2 -8248.471} C_VEL
LIN {X 0,Y 453.507,Z 187.99,A -85,B 0,C 180,E1 -8251.289,E2 -8251.289} C_VEL
LIN {X 0,Y 453.515,Z 187.994,A -85,B 0,C 180,E1 -8254.285,E2 -8254.285} C_VEL
LIN {X 0,Y 453.472,Z 187.994,A -85,B 0,C 180,E1 -8257.204,E2 -8257.204} C_VEL
LIN {X 0,Y 453.497,Z 187.998,A -85,B 0,C 180,E1 -8260.066,E2 -8260.066} C_VEL
LIN {X 0,Y 453.5,Z 187.99,A -85,B 0,C 180,E1 -8262.876,E2 -8262.876} C_VEL
LIN {X 0,Y 453.506,Z 187.994,A -85,B 0,C 180,E1 -8265.644,E2 -8265.644} C_VEL
LIN {X 0,Y 453.553,Z 187.986,A -85,B 0,C 180,E1 -8268.379,E2 -8268.379} C_VEL
LIN {X 0,Y 453.643,Z 187.978,A -85,B 0,C 180,E1 -8271.986,E2 -8271.986} C_VEL
LIN {X 0,Y 453.662,Z 187.97,A -85,B 0,C 180,E1 -8274.667,E2 -8274.667} C_VEL
LIN {X 0,Y 453.735,Z 187.964,A -85,B 0,C 180,E1 -8277.337,E2 -8277.337} C_VEL
LIN {X 0,Y 453.814,Z 187.955,A -85,B 0,C 180,E1 -8280,E2 -8280} C_VEL
LIN {X 0,Y 453.736,Z 187.961,A -85,B 0,C 180,E1 -8282.664,E2 -8282.664} C_VEL
LIN {X 0,Y 453.661,Z 187.972,A -85,B 0,C 180,E1 -8286.226,E2 -8286.226} C_VEL
LIN {X 0,Y 453.583,Z 187.981,A -85,B 0,C 180,E1 -8288.914,E2 -8288.914} C_VEL
LIN {X 0,Y 453.556,Z 187.984,A -85,B 0,C 180,E1 -8292.529,E2 -8292.529} C_VEL
LIN {X 0,Y 453.537,Z 187.986,A -85,B 0,C 180,E1 -8296.197,E2 -8296.197} C_VEL
LIN {X 0,Y 453.513,Z 187.993,A -85,B 0,C 180,E1 -8299.041,E2 -8299.041} C_VEL
LIN {X 0,Y 453.469,Z 187.996,A -85,B 0,C 180,E1 -8301.837,E2 -8301.837} C_VEL
LIN {X 0,Y 453.506,Z 187.991,A -85,B 0,C 180,E1 -8304.735,E2 -8304.735} C_VEL
LIN {X 0,Y 453.525,Z 187.988,A -85,B 0,C 180,E1 -8307.96,E2 -8307.96} C_VEL
LIN {X 0,Y 453.459,Z 187.999,A -85,B 0,C 180,E1 -8311.526,E2 -8311.526} C_VEL
LIN {X 0,Y 453.477,Z 187.997,A -85,B 0,C 180,E1 -8314.777,E2 -8314.777} C_VEL
LIN {X 0,Y 453.458,Z 187.996,A -85,B 0,C 180,E1 -8318.313,E2 -8318.313} C_VEL
LIN {X 0,Y 453.489,Z 187.995,A -85,B 0,C 180,E1 -8320.61,E2 -8320.61} C_VEL
LIN {X 0,Y 453.45,Z 188.001,A -85,B 0,C 180,E1 -8323.245,E2 -8323.245} C_VEL
LIN {X 0,Y 453.459,Z 187.996,A -85,B 0,C 180,E1 -8325.78,E2 -8325.78} C_VEL
LIN {X 0,Y 453.49,Z 187.994,A -85,B 0,C 180,E1 -8329.41,E2 -8329.41} C_VEL
LIN {X 0,Y 453.444,Z 187.999,A -85,B 0,C 180,E1 -8332.229,E2 -8332.229} C_VEL
LIN {X 0,Y 453.485,Z 187.998,A -85,B 0,C 180,E1 -8335.224,E2 -8335.224} C_VEL
LIN {X 0,Y 453.464,Z 188.003,A -85,B 0,C 180,E1 -8338.476,E2 -8338.476} C_VEL
LIN {X 0,Y 453.531,Z 188.124,A -85,B 0,C 180,E1 -8341.949,E2 -8341.949} C_VEL
LIN {X 0,Y 457.145,Z 204.27,A -85,B 0,C 180,E1 -8344.504,E2 -8344.504} C_VEL
LIN {X 0,Y 457.318,Z 208.07,A -85,B 0,C 180,E1 -8345.055,E2 -8345.055} C_VEL
LIN {X 0,Y 456.055,Z 231.425,A -85,B 0,C 180,E1 -8348.295,E2 -8348.295} C_VEL
LIN {X 0,Y 454.898,Z 256.739,A -85,B 0,C 180,E1 -8351.769,E2 -8351.769} C_VEL
LIN {X 0,Y 454.584,Z 264.639,A -85,B 0,C 180,E1 -8352.832,E2 -8352.832} C_VEL
LIN {X 0,Y 455.267,Z 271.45,A -85,B 0,C 180,E1 -8353.007,E2 -8353.007} C_VEL
LIN {X 0,Y 456.729,Z 284.159,A -85,B 0,C 180,E1 -8353.269,E2 -8353.269} C_VEL
LIN {X 0,Y 455.953,Z 373.077,A -85,B 0,C 180,E1 -8354.753,E2 -8354.753} C_VEL
LIN {X 0,Y 455.541,Z 385.992,A -85,B 0,C 180,E1 -8355.139,E2 -8355.139} C_VEL
LIN {X 0,Y 455.101,Z 398.533,A -85,B 0,C 180,E1 -8355.696,E2 -8355.696} C_VEL
LIN {X 0,Y 454.634,Z 409.676,A -85,B 0,C 180,E1 -8356.365,E2 -8356.365} C_VEL
LIN {X 0,Y 454.165,Z 420.49,A -85,B 0,C 180,E1 -8357.192,E2 -8357.192} C_VEL
LIN {X 0,Y 453.686,Z 430.647,A -85,B 0,C 180,E1 -8358.156,E2 -8358.156} C_VEL
LIN {X 0,Y 453.322,Z 440.235,A -85,B 0,C 180,E1 -8359.279,E2 -8359.279} C_VEL
LIN {X 0,Y 452.967,Z 449.431,A -85,B 0,C 180,E1 -8360.625,E2 -8360.625} C_VEL
LIN {X 0,Y 452.814,Z 456.826,A -85,B 0,C 180,E1 -8361.971,E2 -8361.971} C_VEL
LIN {X 0,Y 452.691,Z 463.439,A -85,B 0,C 180,E1 -8363.515,E2 -8363.515} C_VEL
LIN {X 0,Y 452.593,Z 468.54,A -85,B 0,C 180,E1 -8365.101,E2 -8365.101} C_VEL
LIN {X 0,Y 452.717,Z 471.641,A -85,B 0,C 180,E1 -8366.441,E2 -8366.441} C_VEL
LIN {X 0,Y 452.729,Z 473.142,A -85,B 0,C 180,E1 -8367.331,E2 -8367.331} C_VEL
LIN {X 0,Y 452.586,Z 474.782,A -85,B 0,C 180,E1 -8369.111,E2 -8369.111} C_VEL
LIN {X 0,Y 452.607,Z 475,A -85,B 0,C 180,E1 -8370.001,E2 -8370.001} C_VEL
LIN {X 0,Y 452.588,Z 474.764,A -85,B 0,C 180,E1 -8370.89,E2 -8370.89} C_VEL
LIN {X 0,Y 452.733,Z 473.051,A -85,B 0,C 180,E1 -8372.67,E2 -8372.67} C_VEL
LIN {X 0,Y 452.73,Z 471.558,A -85,B 0,C 180,E1 -8373.561,E2 -8373.561} C_VEL
LIN {X 0,Y 452.602,Z 468.429,A -85,B 0,C 180,E1 -8374.9,E2 -8374.9} C_VEL
LIN {X 0,Y 452.692,Z 463.294,A -85,B 0,C 180,E1 -8376.486,E2 -8376.486} C_VEL
LIN {X 0,Y 452.815,Z 456.693,A -85,B 0,C 180,E1 -8378.03,E2 -8378.03} C_VEL
LIN {X 0,Y 452.962,Z 449.343,A -85,B 0,C 180,E1 -8379.377,E2 -8379.377} C_VEL
LIN {X 0,Y 453.343,Z 440.202,A -85,B 0,C 180,E1 -8380.722,E2 -8380.722} C_VEL
LIN {X 0,Y 453.681,Z 430.802,A -85,B 0,C 180,E1 -8381.845,E2 -8381.845} C_VEL
LIN {X 0,Y 454.106,Z 421.543,A -85,B 0,C 180,E1 -8382.75,E2 -8382.75} C_VEL
LIN {X 0,Y 454.612,Z 410.3,A -85,B 0,C 180,E1 -8383.637,E2 -8383.637} C_VEL
LIN {X 0,Y 455.25,Z 397.58,A -85,B 0,C 180,E1 -8384.415,E2 -8384.415} C_VEL
LIN {X 0,Y 455.737,Z 384.402,A -85,B 0,C 180,E1 -8384.999,E2 -8384.999} C_VEL
LIN {X 0,Y 456.151,Z 371.376,A -85,B 0,C 180,E1 -8385.385,E2 -8385.385} C_VEL
LIN {X 0,Y 456.904,Z 283.108,A -85,B 0,C 180,E1 -8386.901,E2 -8386.901} C_VEL
LIN {X 0,Y 454.673,Z 263.532,A -85,B 0,C 180,E1 -8387.366,E2 -8387.366} C_VEL
LIN {X 0,Y 455.527,Z 241.11,A -85,B 0,C 180,E1 -8390.313,E2 -8390.313} C_VEL
LIN {X 0,Y 456.526,Z 218.38,A -85,B 0,C 180,E1 -8393.354,E2 -8393.354} C_VEL
LIN {X 0,Y 457.089,Z 204.031,A -85,B 0,C 180,E1 -8395.305,E2 -8395.305} C_VEL
LIN {X 0,Y 454.495,Z 192.033,A -85,B 0,C 180,E1 -8397.141,E2 -8397.141} C_VEL
LIN {X 0,Y 453.509,Z 188.093,A -85,B 0,C 180,E1 -8397.82,E2 -8397.82} C_VEL
LIN {X 0,Y 453.477,Z 188,A -85,B 0,C 180,E1 -8400.76,E2 -8400.76} C_VEL
LIN {X 0,Y 453.471,Z 187.999,A -85,B 0,C 180,E1 -8403.914,E2 -8403.914} C_VEL
LIN {X 0,Y 453.452,Z 188.004,A -85,B 0,C 180,E1 -8407.19,E2 -8407.19} C_VEL
LIN {X 0,Y 453.473,Z 188,A -85,B 0,C 180,E1 -8410.611,E2 -8410.611} C_VEL
LIN {X 0,Y 453.462,Z 187.998,A -85,B 0,C 180,E1 -8414.222,E2 -8414.222} C_VEL
LIN {X 0,Y 453.451,Z 188.005,A -85,B 0,C 180,E1 -8417.003,E2 -8417.003} C_VEL
LIN {X 0,Y 453.496,Z 187.993,A -85,B 0,C 180,E1 -8419.409,E2 -8419.409} C_VEL
LIN {X 0,Y 453.451,Z 187.998,A -85,B 0,C 180,E1 -8422.227,E2 -8422.227} C_VEL
LIN {X 0,Y 453.485,Z 187.997,A -85,B 0,C 180,E1 -8425.224,E2 -8425.224} C_VEL
LIN {X 0,Y 453.467,Z 187.999,A -85,B 0,C 180,E1 -8428.475,E2 -8428.475} C_VEL
LIN {X 0,Y 453.534,Z 187.99,A -85,B 0,C 180,E1 -8432.04,E2 -8432.04} C_VEL
LIN {X 0,Y 453.502,Z 187.993,A -85,B 0,C 180,E1 -8435.264,E2 -8435.264} C_VEL
LIN {X 0,Y 453.482,Z 188,A -85,B 0,C 180,E1 -8438.415,E2 -8438.415} C_VEL
LIN {X 0,Y 453.524,Z 187.992,A -85,B 0,C 180,E1 -8441.008,E2 -8441.008} C_VEL
LIN {X 0,Y 453.571,Z 187.986,A -85,B 0,C 180,E1 -8443.879,E2 -8443.879} C_VEL
LIN {X 0,Y 453.565,Z 187.984,A -85,B 0,C 180,E1 -8447.471,E2 -8447.471} C_VEL
LIN {X 0,Y 453.587,Z 187.984,A -85,B 0,C 180,E1 -8451.086,E2 -8451.086} C_VEL
LIN {X 0,Y 453.651,Z 187.977,A -85,B 0,C 180,E1 -8453.774,E2 -8453.774} C_VEL
LIN {X 0,Y 453.744,Z 187.967,A -85,B 0,C 180,E1 -8457.336,E2 -8457.336} C_VEL
LIN {X 0,Y 453.721,Z 188.139,A -85,B 0,C 180,E1 -8458.585,E2 -8458.585} C_VEL
LIN {X 0,Y 454.737,Z 193.237,A -85,B 0,C 180,E1 -8459.557,E2 -8459.557} C_VEL
LIN {X 0,Y 454.567,Z 209.677,A -85,B 0,C 180,E1 -8462.436,E2 -8462.436} C_VEL
LIN {X 0,Y 454.462,Z 227.839,A -85,B 0,C 180,E1 -8465.657,E2 -8465.657} C_VEL
LIN {X 0,Y 455.911,Z 235.262,A -85,B 0,C 180,E1 -8465.903,E2 -8465.903} C_VEL
LIN {X 0,Y 456.881,Z 241.508,A -85,B 0,C 180,E1 -8466.07,E2 -8466.07} C_VEL
LIN {X 0,Y 455.862,Z 310.761,A -85,B 0,C 180,E1 -8467.418,E2 -8467.418} C_VEL
LIN {X 0,Y 455.733,Z 322.135,A -85,B 0,C 180,E1 -8467.81,E2 -8467.81} C_VEL
LIN {X 0,Y 455.396,Z 333.914,A -85,B 0,C 180,E1 -8468.409,E2 -8468.409} C_VEL
LIN {X 0,Y 455.076,Z 344.037,A -85,B 0,C 180,E1 -8469.108,E2 -8469.108} C_VEL
LIN {X 0,Y 454.707,Z 354.195,A -85,B 0,C 180,E1 -8470.013,E2 -8470.013} C_VEL
LIN {X 0,Y 454.319,Z 362.251,A -85,B 0,C 180,E1 -8470.923,E2 -8470.923} C_VEL
LIN {X 0,Y 453.932,Z 370.347,A -85,B 0,C 180,E1 -8472.064,E2 -8472.064} C_VEL
LIN {X 0,Y 453.619,Z 376.612,A -85,B 0,C 180,E1 -8473.187,E2 -8473.187} C_VEL
LIN {X 0,Y 453.36,Z 381.803,A -85,B 0,C 180,E1 -8474.361,E2 -8474.361} C_VEL
LIN {X 0,Y 453.181,Z 385.023,A -85,B 0,C 180,E1 -8475.286,E2 -8475.286} C_VEL
LIN {X 0,Y 453.072,Z 387.591,A -85,B 0,C 180,E1 -8476.213,E2 -8476.213} C_VEL
LIN {X 0,Y 452.957,Z 389.561,A -85,B 0,C 180,E1 -8477.145,E2 -8477.145} C_VEL
LIN {X 0,Y 452.834,Z 390.915,A -85,B 0,C 180,E1 -8478.083,E2 -8478.083} C_VEL
LIN {X 0,Y 452.787,Z 391.709,A -85,B 0,C 180,E1 -8479.023,E2 -8479.023} C_VEL
LIN {X 0,Y 452.749,Z 391.947,A -85,B 0,C 180,E1 -8479.968,E2 -8479.968} C_VEL
LIN {X 0,Y 452.772,Z 391.22,A -85,B 0,C 180,E1 -8481.357,E2 -8481.357} C_VEL
LIN {X 0,Y 452.849,Z 389.121,A -85,B 0,C 180,E1 -8482.829,E2 -8482.829} C_VEL
LIN {X 0,Y 453.051,Z 385.579,A -85,B 0,C 180,E1 -8484.272,E2 -8484.272} C_VEL
LIN {X 0,Y 453.216,Z 380.403,A -85,B 0,C 180,E1 -8485.734,E2 -8485.734} C_VEL
LIN {X 0,Y 453.426,Z 374.613,A -85,B 0,C 180,E1 -8486.959,E2 -8486.959} C_VEL
LIN {X 0,Y 453.694,Z 368.425,A -85,B 0,C 180,E1 -8487.998,E2 -8487.998} C_VEL
LIN {X 0,Y 454.02,Z 359.552,A -85,B 0,C 180,E1 -8489.183,E2 -8489.183} C_VEL
LIN {X 0,Y 454.403,Z 350.084,A -85,B 0,C 180,E1 -8490.167,E2 -8490.167} C_VEL
LIN {X 0,Y 454.731,Z 340.958,A -85,B 0,C 180,E1 -8490.923,E2 -8490.923} C_VEL
LIN {X 0,Y 455.042,Z 329.026,A -85,B 0,C 180,E1 -8491.676,E2 -8491.676} C_VEL
LIN {X 0,Y 455.29,Z 316.714,A -85,B 0,C 180,E1 -8492.221,E2 -8492.221} C_VEL
LIN {X 0,Y 455.427,Z 304.408,A -85,B 0,C 180,E1 -8492.562,E2 -8492.562} C_VEL
LIN {X 0,Y 456.051,Z 239.047,A -85,B 0,C 180,E1 -8493.72,E2 -8493.72} C_VEL
LIN {X 0,Y 454.011,Z 227.246,A -85,B 0,C 180,E1 -8494.022,E2 -8494.022} C_VEL
LIN {X 0,Y 453.97,Z 226.275,A -85,B 0,C 180,E1 -8494.138,E2 -8494.138} C_VEL
LIN {X 0,Y 454.311,Z 210.051,A -85,B 0,C 180,E1 -8497.381,E2 -8497.381} C_VEL
LIN {X 0,Y 454.605,Z 194.805,A -85,B 0,C 180,E1 -8500.488,E2 -8500.488} C_VEL
LIN {X 0,Y 453.537,Z 188.17,A -85,B 0,C 180,E1 -8501.943,E2 -8501.943} C_VEL
LIN {X 0,Y 453.483,Z 187.999,A -85,B 0,C 180,E1 -8505.471,E2 -8505.471} C_VEL
LIN {X 0,Y 453.478,Z 187.997,A -85,B 0,C 180,E1 -8508.209,E2 -8508.209} C_VEL
LIN {X 0,Y 453.485,Z 187.992,A -85,B 0,C 180,E1 -8510.794,E2 -8510.794} C_VEL
LIN {X 0,Y 453.453,Z 188.003,A -85,B 0,C 180,E1 -8513.784,E2 -8513.784} C_VEL
LIN {X 0,Y 452.799,Z 188.079,A -85,B 0,C 180,E1 -8514.525,E2 -8514.525} C_VEL
LIN {X 0,Y 449.962,Z 188.439,A -85,B 0,C 180,E1 -8515.729,E2 -8515.729} C_VEL
LIN {X 0,Y 447.551,Z 188.744,A -85,B 0,C 180,E1 -8516.7,E2 -8516.7} C_VEL
LIN {X 0,Y 446.507,Z 188.871,A -85,B 0,C 180,E1 -8517.451,E2 -8517.451} C_VEL
LIN {X 0,Y 446.418,Z 188.879,A -85,B 0,C 180,E1 -8517.705,E2 -8517.705} C_VEL
LIN {X 0,Y 446.447,Z 188.87,A -85,B 0,C 180,E1 -8520.79,E2 -8520.79} C_VEL
LIN {X 0,Y 446.476,Z 188.869,A -85,B 0,C 180,E1 -8523.848,E2 -8523.848} C_VEL
LIN {X 0,Y 446.427,Z 188.873,A -85,B 0,C 180,E1 -8526.823,E2 -8526.823} C_VEL
LIN {X 0,Y 446.442,Z 188.873,A -85,B 0,C 180,E1 -8529.737,E2 -8529.737} C_VEL
LIN {X 0,Y 446.461,Z 188.868,A -85,B 0,C 180,E1 -8532.597,E2 -8532.597} C_VEL
LIN {X 0,Y 446.47,Z 188.873,A -85,B 0,C 180,E1 -8535.412,E2 -8535.412} C_VEL
LIN {X 0,Y 446.516,Z 188.861,A -85,B 0,C 180,E1 -8538.193,E2 -8538.193} C_VEL
LIN {X 0,Y 446.598,Z 188.851,A -85,B 0,C 180,E1 -8541.857,E2 -8541.857} C_VEL
LIN {X 0,Y 446.645,Z 188.846,A -85,B 0,C 180,E1 -8544.582,E2 -8544.582} C_VEL
LIN {X 0,Y 446.706,Z 188.842,A -85,B 0,C 180,E1 -8547.294,E2 -8547.294} C_VEL
LIN {X 0,Y 446.792,Z 188.826,A -85,B 0,C 180,E1 -8549.999,E2 -8549.999} C_VEL
LIN {X 0,Y 446.706,Z 188.84,A -85,B 0,C 180,E1 -8552.705,E2 -8552.705} C_VEL
LIN {X 0,Y 446.636,Z 188.847,A -85,B 0,C 180,E1 -8556.323,E2 -8556.323} C_VEL
LIN {X 0,Y 446.534,Z 188.865,A -85,B 0,C 180,E1 -8559.055,E2 -8559.055} C_VEL
LIN {X 0,Y 446.517,Z 188.866,A -85,B 0,C 180,E1 -8562.729,E2 -8562.729} C_VEL
LIN {X 0,Y 446.492,Z 188.865,A -85,B 0,C 180,E1 -8566.227,E2 -8566.227} C_VEL
LIN {X 0,Y 446.465,Z 188.869,A -85,B 0,C 180,E1 -8569.303,E2 -8569.303} C_VEL
LIN {X 0,Y 446.413,Z 188.875,A -85,B 0,C 180,E1 -8572.199,E2 -8572.199} C_VEL
LIN {X 0,Y 446.453,Z 188.871,A -85,B 0,C 180,E1 -8575.152,E2 -8575.152} C_VEL
LIN {X 0,Y 446.478,Z 188.868,A -85,B 0,C 180,E1 -8578.178,E2 -8578.178} C_VEL
LIN {X 0,Y 446.414,Z 188.874,A -85,B 0,C 180,E1 -8581.775,E2 -8581.775} C_VEL
LIN {X 0,Y 446.434,Z 188.879,A -85,B 0,C 180,E1 -8584.521,E2 -8584.521} C_VEL
LIN {X 0,Y 446.429,Z 188.874,A -85,B 0,C 180,E1 -8588.082,E2 -8588.082} C_VEL
LIN {X 0,Y 446.44,Z 188.872,A -85,B 0,C 180,E1 -8590.92,E2 -8590.92} C_VEL
LIN {X 0,Y 446.437,Z 188.872,A -85,B 0,C 180,E1 -8593.84,E2 -8593.84} C_VEL
LIN {X 0,Y 446.407,Z 188.882,A -85,B 0,C 180,E1 -8596.401,E2 -8596.401} C_VEL
LIN {X 0,Y 446.459,Z 188.87,A -85,B 0,C 180,E1 -8599.804,E2 -8599.804} C_VEL
LIN {X 0,Y 446.424,Z 188.878,A -85,B 0,C 180,E1 -8602.123,E2 -8602.123} C_VEL
LIN {X 0,Y 446.422,Z 188.873,A -85,B 0,C 180,E1 -8605.477,E2 -8605.477} C_VEL
LIN {X 0,Y 446.422,Z 188.874,A -85,B 0,C 180,E1 -8608.701,E2 -8608.701} C_VEL
LIN {X 0,Y 446.476,Z 188.87,A -85,B 0,C 180,E1 -8611.821,E2 -8611.821} C_VEL
LIN {X 0,Y 446.449,Z 188.869,A -85,B 0,C 180,E1 -8614.848,E2 -8614.848} C_VEL
LIN {X 0,Y 446.439,Z 188.875,A -85,B 0,C 180,E1 -8618.245,E2 -8618.245} C_VEL
LIN {X 0,Y 446.449,Z 188.873,A -85,B 0,C 180,E1 -8621.649,E2 -8621.649} C_VEL
LIN {X 0,Y 446.507,Z 188.863,A -85,B 0,C 180,E1 -8624.48,E2 -8624.48} C_VEL
LIN {X 0,Y 446.51,Z 188.865,A -85,B 0,C 180,E1 -8628.193,E2 -8628.193} C_VEL
LIN {X 0,Y 446.592,Z 188.858,A -85,B 0,C 180,E1 -8631.858,E2 -8631.858} C_VEL
LIN {X 0,Y 446.636,Z 188.846,A -85,B 0,C 180,E1 -8634.583,E2 -8634.583} C_VEL
LIN {X 0,Y 446.655,Z 188.845,A -85,B 0,C 180,E1 -8638.197,E2 -8638.197} C_VEL
LIN {X 0,Y 446.785,Z 188.831,A -85,B 0,C 180,E1 -8640,E2 -8640} C_VEL
LIN {X 0,Y 446.683,Z 188.84,A -85,B 0,C 180,E1 -8642.706,E2 -8642.706} C_VEL
LIN {X 0,Y 446.63,Z 188.847,A -85,B 0,C 180,E1 -8646.324,E2 -8646.324} C_VEL
LIN {X 0,Y 446.529,Z 188.861,A -85,B 0,C 180,E1 -8649.056,E2 -8649.056} C_VEL
LIN {X 0,Y 446.514,Z 188.861,A -85,B 0,C 180,E1 -8652.73,E2 -8652.73} C_VEL
LIN {X 0,Y 446.489,Z 188.864,A -85,B 0,C 180,E1 -8656.228,E2 -8656.228} C_VEL
LIN {X 0,Y 446.462,Z 188.874,A -85,B 0,C 180,E1 -8659.304,E2 -8659.304} C_VEL
LIN {X 0,Y 446.411,Z 188.874,A -85,B 0,C 180,E1 -8662.2,E2 -8662.2} C_VEL
LIN {X 0,Y 446.451,Z 188.875,A -85,B 0,C 180,E1 -8665.153,E2 -8665.153} C_VEL
LIN {X 0,Y 446.479,Z 188.865,A -85,B 0,C 180,E1 -8668.179,E2 -8668.179} C_VEL
LIN {X 0,Y 446.412,Z 188.875,A -85,B 0,C 180,E1 -8671.776,E2 -8671.776} C_VEL
LIN {X 0,Y 446.417,Z 188.874,A -85,B 0,C 180,E1 -8674.525,E2 -8674.525} C_VEL
LIN {X 0,Y 446.409,Z 188.874,A -85,B 0,C 180,E1 -8678.08,E2 -8678.08} C_VEL
LIN {X 0,Y 446.423,Z 188.879,A -85,B 0,C 180,E1 -8680.919,E2 -8680.919} C_VEL
LIN {X 0,Y 446.396,Z 188.876,A -85,B 0,C 180,E1 -8683.847,E2 -8683.847} C_VEL
LIN {X 0,Y 446.395,Z 188.877,A -85,B 0,C 180,E1 -8686.404,E2 -8686.404} C_VEL
LIN {X 0,Y 446.438,Z 188.87,A -85,B 0,C 180,E1 -8689.803,E2 -8689.803} C_VEL
LIN {X 0,Y 446.397,Z 188.88,A -85,B 0,C 180,E1 -8693.256,E2 -8693.256} C_VEL
LIN {X 0,Y 446.447,Z 188.876,A -85,B 0,C 180,E1 -8696.567,E2 -8696.567} C_VEL
LIN {X 0,Y 446.427,Z 188.877,A -85,B 0,C 180,E1 -8699.981,E2 -8699.981} C_VEL
LIN {X 0,Y 446.502,Z 189.022,A -85,B 0,C 180,E1 -8701.709,E2 -8701.709} C_VEL
LIN {X 0,Y 450.115,Z 205.114,A -85,B 0,C 180,E1 -8704.291,E2 -8704.291} C_VEL
LIN {X 0,Y 450.452,Z 208.603,A -85,B 0,C 180,E1 -8704.814,E2 -8704.814} C_VEL
LIN {X 0,Y 449.194,Z 230.802,A -85,B 0,C 180,E1 -8707.946,E2 -8707.946} C_VEL
LIN {X 0,Y 447.969,Z 256.119,A -85,B 0,C 180,E1 -8711.477,E2 -8711.477} C_VEL
LIN {X 0,Y 447.612,Z 264.48,A -85,B 0,C 180,E1 -8712.615,E2 -8712.615} C_VEL
LIN {X 0,Y 449.58,Z 282.274,A -85,B 0,C 180,E1 -8713.016,E2 -8713.016} C_VEL
LIN {X 0,Y 449.763,Z 291.195,A -85,B 0,C 180,E1 -8713.176,E2 -8713.176} C_VEL
LIN {X 0,Y 448.992,Z 372.828,A -85,B 0,C 180,E1 -8714.569,E2 -8714.569} C_VEL
LIN {X 0,Y 448.56,Z 386.418,A -85,B 0,C 180,E1 -8714.989,E2 -8714.989} C_VEL
LIN {X 0,Y 448.082,Z 399.152,A -85,B 0,C 180,E1 -8715.583,E2 -8715.583} C_VEL
LIN {X 0,Y 447.547,Z 411.652,A -85,B 0,C 180,E1 -8716.377,E2 -8716.377} C_VEL
LIN {X 0,Y 447.107,Z 422.786,A -85,B 0,C 180,E1 -8717.288,E2 -8717.288} C_VEL
LIN {X 0,Y 446.532,Z 431.757,A -85,B 0,C 180,E1 -8718.194,E2 -8718.194} C_VEL
LIN {X 0,Y 446.213,Z 440.99,A -85,B 0,C 180,E1 -8719.336,E2 -8719.336} C_VEL
LIN {X 0,Y 445.851,Z 449.958,A -85,B 0,C 180,E1 -8720.703,E2 -8720.703} C_VEL
LIN {X 0,Y 445.699,Z 457.099,A -85,B 0,C 180,E1 -8722.07,E2 -8722.07} C_VEL
LIN {X 0,Y 445.579,Z 463.591,A -85,B 0,C 180,E1 -8723.662,E2 -8723.662} C_VEL
LIN {X 0,Y 445.527,Z 467.818,A -85,B 0,C 180,E1 -8725.023,E2 -8725.023} C_VEL
LIN {X 0,Y 445.643,Z 470.942,A -85,B 0,C 180,E1 -8726.384,E2 -8726.384} C_VEL
LIN {X 0,Y 445.674,Z 472.462,A -85,B 0,C 180,E1 -8727.289,E2 -8727.289} C_VEL
LIN {X 0,Y 445.555,Z 473.492,A -85,B 0,C 180,E1 -8728.193,E2 -8728.193} C_VEL
LIN {X 0,Y 445.518,Z 474.117,A -85,B 0,C 180,E1 -8729.097,E2 -8729.097} C_VEL
LIN {X 0,Y 445.537,Z 474.341,A -85,B 0,C 180,E1 -8730.001,E2 -8730.001} C_VEL
LIN {X 0,Y 445.519,Z 474.116,A -85,B 0,C 180,E1 -8730.904,E2 -8730.904} C_VEL
LIN {X 0,Y 445.679,Z 472.406,A -85,B 0,C 180,E1 -8732.712,E2 -8732.712} C_VEL
LIN {X 0,Y 445.655,Z 470.914,A -85,B 0,C 180,E1 -8733.617,E2 -8733.617} C_VEL
LIN {X 0,Y 445.535,Z 467.785,A -85,B 0,C 180,E1 -8734.978,E2 -8734.978} C_VEL
LIN {X 0,Y 445.606,Z 463.085,A -85,B 0,C 180,E1 -8736.472,E2 -8736.472} C_VEL
LIN {X 0,Y 445.699,Z 457.097,A -85,B 0,C 180,E1 -8737.931,E2 -8737.931} C_VEL
LIN {X 0,Y 445.848,Z 450.039,A -85,B 0,C 180,E1 -8739.299,E2 -8739.299} C_VEL
LIN {X 0,Y 446.117,Z 442.839,A -85,B 0,C 180,E1 -8740.438,E2 -8740.438} C_VEL
LIN {X 0,Y 446.481,Z 434.15,A -85,B 0,C 180,E1 -8741.578,E2 -8741.578} C_VEL
LIN {X 0,Y 447.048,Z 423.414,A -85,B 0,C 180,E1 -8742.715,E2 -8742.715} C_VEL
LIN {X 0,Y 447.53,Z 412.767,A -85,B 0,C 180,E1 -8743.625,E2 -8743.625} C_VEL
LIN {X 0,Y 448.153,Z 400.978,A -85,B 0,C 180,E1 -8744.416,E2 -8744.416} C_VEL
LIN {X 0,Y 448.701,Z 388.703,A -85,B 0,C 180,E1 -8745.036,E2 -8745.036} C_VEL
LIN {X 0,Y 449.146,Z 376.211,A -85,B 0,C 180,E1 -8745.485,E2 -8745.485} C_VEL
LIN {X 0,Y 449.438,Z 361.843,A -85,B 0,C 180,E1 -8745.795,E2 -8745.795} C_VEL
LIN {X 0,Y 450.213,Z 284.509,A -85,B 0,C 180,E1 -8747.137,E2 -8747.137} C_VEL
LIN {X 0,Y 447.747,Z 263.314,A -85,B 0,C 180,E1 -8747.643,E2 -8747.643} C_VEL
LIN {X 0,Y 448.592,Z 242.57,A -85,B 0,C 180,E1 -8750.401,E2 -8750.401} C_VEL
LIN {X 0,Y 449.669,Z 219.925,A -85,B 0,C 180,E1 -8753.488,E2 -8753.488} C_VEL
LIN {X 0,Y 450.258,Z 205.687,A -85,B 0,C 180,E1 -8755.451,E2 -8755.451} C_VEL
LIN {X 0,Y 447.657,Z 193.64,A -85,B 0,C 180,E1 -8757.337,E2 -8757.337} C_VEL
LIN {X 0,Y 446.463,Z 189.007,A -85,B 0,C 180,E1 -8758.129,E2 -8758.129} C_VEL
LIN {X 0,Y 446.418,Z 188.88,A -85,B 0,C 180,E1 -8761.301,E2 -8761.301} C_VEL
LIN {X 0,Y 446.426,Z 188.878,A -85,B 0,C 180,E1 -8764.524,E2 -8764.524} C_VEL
LIN {X 0,Y 446.413,Z 188.876,A -85,B 0,C 180,E1 -8768.078,E2 -8768.078} C_VEL
LIN {X 0,Y 446.409,Z 188.881,A -85,B 0,C 180,E1 -8771.394,E2 -8771.394} C_VEL
LIN {X 0,Y 446.453,Z 188.876,A -85,B 0,C 180,E1 -8775.104,E2 -8775.104} C_VEL
LIN {X 0,Y 446.421,Z 188.876,A -85,B 0,C 180,E1 -8778.608,E2 -8778.608} C_VEL
LIN {X 0,Y 446.442,Z 188.878,A -85,B 0,C 180,E1 -8780.972,E2 -8780.972} C_VEL
LIN {X 0,Y 446.42,Z 188.875,A -85,B 0,C 180,E1 -8784.374,E2 -8784.374} C_VEL
LIN {X 0,Y 446.422,Z 188.874,A -85,B 0,C 180,E1 -8787.638,E2 -8787.638} C_VEL
LIN {X 0,Y 446.449,Z 188.873,A -85,B 0,C 180,E1 -8790.79,E2 -8790.79} C_VEL
LIN {X 0,Y 446.48,Z 188.867,A -85,B 0,C 180,E1 -8793.848,E2 -8793.848} C_VEL
LIN {X 0,Y 446.428,Z 188.876,A -85,B 0,C 180,E1 -8796.823,E2 -8796.823} C_VEL
LIN {X 0,Y 446.445,Z 188.872,A -85,B 0,C 180,E1 -8799.737,E2 -8799.737} C_VEL
LIN {X 0,Y 446.457,Z 188.874,A -85,B 0,C 180,E1 -8802.596,E2 -8802.596} C_VEL
LIN {X 0,Y 446.47,Z 188.869,A -85,B 0,C 180,E1 -8805.412,E2 -8805.412} C_VEL
LIN {X 0,Y 446.519,Z 188.867,A -85,B 0,C 180,E1 -8808.193,E2 -8808.193} C_VEL
LIN {X 0,Y 446.534,Z 188.863,A -85,B 0,C 180,E1 -8810.944,E2 -8810.944} C_VEL
LIN {X 0,Y 446.619,Z 188.853,A -85,B 0,C 180,E1 -8813.675,E2 -8813.675} C_VEL
LIN {X 0,Y 446.691,Z 188.846,A -85,B 0,C 180,E1 -8817.294,E2 -8817.294} C_VEL
LIN {X 0,Y 446.695,Z 189.059,A -85,B 0,C 180,E1 -8818.309,E2 -8818.309} C_VEL
LIN {X 0,Y 447.911,Z 195.534,A -85,B 0,C 180,E1 -8819.55,E2 -8819.55} C_VEL
LIN {X 0,Y 447.669,Z 213.299,A -85,B 0,C 180,E1 -8822.699,E2 -8822.699} C_VEL
LIN {X 0,Y 447.557,Z 228.087,A -85,B 0,C 180,E1 -8825.349,E2 -8825.349} C_VEL
LIN {X 0,Y 448.402,Z 232.365,A -85,B 0,C 180,E1 -8825.523,E2 -8825.523} C_VEL
LIN {X 0,Y 450.144,Z 242.025,A -85,B 0,C 180,E1 -8825.796,E2 -8825.796} C_VEL
LIN {X 0,Y 449.04,Z 310.678,A -85,B 0,C 180,E1 -8827.164,E2 -8827.164} C_VEL
LIN {X 0,Y 448.885,Z 322.879,A -85,B 0,C 180,E1 -8827.591,E2 -8827.591} C_VEL
LIN {X 0,Y 448.545,Z 334.361,A -85,B 0,C 180,E1 -8828.186,E2 -8828.186} C_VEL
LIN {X 0,Y 448.178,Z 344.746,A -85,B 0,C 180,E1 -8828.915,E2 -8828.915} C_VEL
LIN {X 0,Y 447.809,Z 354.804,A -85,B 0,C 180,E1 -8829.827,E2 -8829.827} C_VEL
LIN {X 0,Y 447.339,Z 363.784,A -85,B 0,C 180,E1 -8830.866,E2 -8830.866} C_VEL
LIN {X 0,Y 446.931,Z 371.614,A -85,B 0,C 180,E1 -8832.015,E2 -8832.015} C_VEL
LIN {X 0,Y 446.609,Z 377.72,A -85,B 0,C 180,E1 -8833.143,E2 -8833.143} C_VEL
LIN {X 0,Y 446.282,Z 383.742,A -85,B 0,C 180,E1 -8834.593,E2 -8834.593} C_VEL
LIN {X 0,Y 446.036,Z 388.029,A -85,B 0,C 180,E1 -8836.023,E2 -8836.023} C_VEL
LIN {X 0,Y 445.859,Z 390.794,A -85,B 0,C 180,E1 -8837.427,E2 -8837.427} C_VEL
LIN {X 0,Y 445.743,Z 392.347,A -85,B 0,C 180,E1 -8838.912,E2 -8838.912} C_VEL
LIN {X 0,Y 445.698,Z 392.528,A -85,B 0,C 180,E1 -8840.298,E2 -8840.298} C_VEL
LIN {X 0,Y 445.707,Z 391.714,A -85,B 0,C 180,E1 -8841.514,E2 -8841.514} C_VEL
LIN {X 0,Y 445.746,Z 390.804,A -85,B 0,C 180,E1 -8842.234,E2 -8842.234} C_VEL
LIN {X 0,Y 445.831,Z 389.011,A -85,B 0,C 180,E1 -8843.209,E2 -8843.209} C_VEL
LIN {X 0,Y 446.015,Z 385.088,A -85,B 0,C 180,E1 -8844.681,E2 -8844.681} C_VEL
LIN {X 0,Y 446.228,Z 379.454,A -85,B 0,C 180,E1 -8846.167,E2 -8846.167} C_VEL
LIN {X 0,Y 446.479,Z 373.159,A -85,B 0,C 180,E1 -8847.414,E2 -8847.414} C_VEL
LIN {X 0,Y 446.817,Z 365.423,A -85,B 0,C 180,E1 -8848.616,E2 -8848.616} C_VEL
LIN {X 0,Y 447.194,Z 356.846,A -85,B 0,C 180,E1 -8849.672,E2 -8849.672} C_VEL
LIN {X 0,Y 447.563,Z 346.9,A -85,B 0,C 180,E1 -8850.634,E2 -8850.634} C_VEL
LIN {X 0,Y 447.883,Z 337.98,A -85,B 0,C 180,E1 -8851.317,E2 -8851.317} C_VEL
LIN {X 0,Y 448.165,Z 327.161,A -85,B 0,C 180,E1 -8851.955,E2 -8851.955} C_VEL
LIN {X 0,Y 448.337,Z 315.324,A -85,B 0,C 180,E1 -8852.455,E2 -8852.455} C_VEL
LIN {X 0,Y 448.502,Z 303.832,A -85,B 0,C 180,E1 -8852.758,E2 -8852.758} C_VEL
LIN {X 0,Y 449.151,Z 239.793,A -85,B 0,C 180,E1 -8853.922,E2 -8853.922} C_VEL
LIN {X 0,Y 446.984,Z 227.198,A -85,B 0,C 180,E1 -8854.254,E2 -8854.254} C_VEL
LIN {X 0,Y 447.291,Z 212.272,A -85,B 0,C 180,E1 -8857.222,E2 -8857.222} C_VEL
LIN {X 0,Y 447.626,Z 196.954,A -85,B 0,C 180,E1 -8860.364,E2 -8860.364} C_VEL
LIN {X 0,Y 446.882,Z 190.891,A -85,B 0,C 180,E1 -8861.667,E2 -8861.667} C_VEL
LIN {X 0,Y 446.502,Z 188.9,A -85,B 0,C 180,E1 -8862.169,E2 -8862.169} C_VEL
LIN {X 0,Y 446.45,Z 188.874,A -85,B 0,C 180,E1 -8865.103,E2 -8865.103} C_VEL
LIN {X 0,Y 446.427,Z 188.872,A -85,B 0,C 180,E1 -8868.608,E2 -8868.608} C_VEL
LIN {X 0,Y 446.436,Z 188.871,A -85,B 0,C 180,E1 -8870.972,E2 -8870.972} C_VEL
LIN {X 0,Y 446.419,Z 188.873,A -85,B 0,C 180,E1 -8874.374,E2 -8874.374} C_VEL
LIN {X 0,Y 446.418,Z 188.879,A -85,B 0,C 180,E1 -8877.705,E2 -8877.705} C_VEL
LIN {X 0,Y 445.747,Z 188.957,A -85,B 0,C 180,E1 -8878.458,E2 -8878.458} C_VEL
LIN {X 0,Y 442.923,Z 189.314,A -85,B 0,C 180,E1 -8879.683,E2 -8879.683} C_VEL
LIN {X 0,Y 440.539,Z 189.616,A -85,B 0,C 180,E1 -8880.671,E2 -8880.671} C_VEL
LIN {X 0,Y 439.513,Z 189.741,A -85,B 0,C 180,E1 -8881.434,E2 -8881.434} C_VEL
LIN {X 0,Y 439.428,Z 189.749,A -85,B 0,C 180,E1 -8881.692,E2 -8881.692} C_VEL
LIN {X 0,Y 439.404,Z 189.747,A -85,B 0,C 180,E1 -8884.415,E2 -8884.415} C_VEL
LIN {X 0,Y 439.363,Z 189.76,A -85,B 0,C 180,E1 -8887.424,E2 -8887.424} C_VEL
LIN {X 0,Y 439.44,Z 189.743,A -85,B 0,C 180,E1 -8890.662,E2 -8890.662} C_VEL
LIN {X 0,Y 439.461,Z 189.739,A -85,B 0,C 180,E1 -8894.224,E2 -8894.224} C_VEL
LIN {X 0,Y 439.482,Z 189.737,A -85,B 0,C 180,E1 -8898.001,E2 -8898.001} C_VEL
LIN {X 0,Y 439.546,Z 189.731,A -85,B 0,C 180,E1 -8901.726,E2 -8901.726} C_VEL
LIN {X 0,Y 439.62,Z 189.72,A -85,B 0,C 180,E1 -8904.495,E2 -8904.495} C_VEL
LIN {X 0,Y 439.633,Z 189.718,A -85,B 0,C 180,E1 -8908.167,E2 -8908.167} C_VEL
LIN {X 0,Y 439.762,Z 189.702,A -85,B 0,C 180,E1 -8909.999,E2 -8909.999} C_VEL
LIN {X 0,Y 439.653,Z 189.72,A -85,B 0,C 180,E1 -8912.748,E2 -8912.748} C_VEL
LIN {X 0,Y 439.608,Z 189.723,A -85,B 0,C 180,E1 -8916.425,E2 -8916.425} C_VEL
LIN {X 0,Y 439.496,Z 189.739,A -85,B 0,C 180,E1 -8919.201,E2 -8919.201} C_VEL
LIN {X 0,Y 439.461,Z 189.747,A -85,B 0,C 180,E1 -8922.937,E2 -8922.937} C_VEL
LIN {X 0,Y 439.443,Z 189.744,A -85,B 0,C 180,E1 -8926.348,E2 -8926.348} C_VEL
LIN {X 0,Y 439.398,Z 189.747,A -85,B 0,C 180,E1 -8929.626,E2 -8929.626} C_VEL
LIN {X 0,Y 439.36,Z 189.758,A -85,B 0,C 180,E1 -8932.575,E2 -8932.575} C_VEL
LIN {X 0,Y 439.4,Z 189.747,A -85,B 0,C 180,E1 -8935.584,E2 -8935.584} C_VEL
LIN {X 0,Y 439.411,Z 189.753,A -85,B 0,C 180,E1 -8938.673,E2 -8938.673} C_VEL
LIN {X 0,Y 439.364,Z 189.753,A -85,B 0,C 180,E1 -8942.03,E2 -8942.03} C_VEL
LIN {X 0,Y 439.395,Z 189.748,A -85,B 0,C 180,E1 -8945.341,E2 -8945.341} C_VEL
LIN {X 0,Y 439.388,Z 189.755,A -85,B 0,C 180,E1 -8948.593,E2 -8948.593} C_VEL
LIN {X 0,Y 439.397,Z 189.748,A -85,B 0,C 180,E1 -8951.259,E2 -8951.259} C_VEL
LIN {X 0,Y 439.401,Z 189.75,A -85,B 0,C 180,E1 -8954.728,E2 -8954.728} C_VEL
LIN {X 0,Y 439.389,Z 189.75,A -85,B 0,C 180,E1 -8957.796,E2 -8957.796} C_VEL
LIN {X 0,Y 439.441,Z 189.749,A -85,B 0,C 180,E1 -8960.23,E2 -8960.23} C_VEL
LIN {X 0,Y 439.369,Z 189.753,A -85,B 0,C 180,E1 -8963.713,E2 -8963.713} C_VEL
LIN {X 0,Y 439.367,Z 189.751,A -85,B 0,C 180,E1 -8967.054,E2 -8967.054} C_VEL
LIN {X 0,Y 439.388,Z 189.755,A -85,B 0,C 180,E1 -8970.275,E2 -8970.275} C_VEL
LIN {X 0,Y 439.424,Z 189.746,A -85,B 0,C 180,E1 -8973.589,E2 -8973.589} C_VEL
LIN {X 0,Y 439.378,Z 189.753,A -85,B 0,C 180,E1 -8976.43,E2 -8976.43} C_VEL
LIN {X 0,Y 439.38,Z 189.751,A -85,B 0,C 180,E1 -8979.397,E2 -8979.397} C_VEL
LIN {X 0,Y 439.424,Z 189.747,A -85,B 0,C 180,E1 -8982.31,E2 -8982.31} C_VEL
LIN {X 0,Y 439.443,Z 189.742,A -85,B 0,C 180,E1 -8985.174,E2 -8985.174} C_VEL
LIN {X 0,Y 439.476,Z 189.744,A -85,B 0,C 180,E1 -8988.002,E2 -8988.002} C_VEL
LIN {X 0,Y 439.539,Z 189.737,A -85,B 0,C 180,E1 -8991.727,E2 -8991.727} C_VEL
LIN {X 0,Y 439.612,Z 189.721,A -85,B 0,C 180,E1 -8994.496,E2 -8994.496} C_VEL
LIN {X 0,Y 439.625,Z 189.721,A -85,B 0,C 180,E1 -8998.168,E2 -8998.168} C_VEL
LIN {X 0,Y 439.755,Z 189.706,A -85,B 0,C 180,E1 -9000,E2 -9000} C_VEL
LIN {X 0,Y 439.633,Z 189.718,A -85,B 0,C 180,E1 -9002.749,E2 -9002.749} C_VEL
LIN {X 0,Y 439.605,Z 189.722,A -85,B 0,C 180,E1 -9006.426,E2 -9006.426} C_VEL
LIN {X 0,Y 439.491,Z 189.739,A -85,B 0,C 180,E1 -9009.202,E2 -9009.202} C_VEL
LIN {X 0,Y 439.458,Z 189.742,A -85,B 0,C 180,E1 -9012.938,E2 -9012.938} C_VEL
LIN {X 0,Y 439.44,Z 189.742,A -85,B 0,C 180,E1 -9016.349,E2 -9016.349} C_VEL
LIN {X 0,Y 439.395,Z 189.752,A -85,B 0,C 180,E1 -9019.627,E2 -9019.627} C_VEL
LIN {X 0,Y 439.358,Z 189.753,A -85,B 0,C 180,E1 -9022.576,E2 -9022.576} C_VEL
LIN {X 0,Y 439.399,Z 189.751,A -85,B 0,C 180,E1 -9025.586,E2 -9025.586} C_VEL
LIN {X 0,Y 439.411,Z 189.747,A -85,B 0,C 180,E1 -9028.674,E2 -9028.674} C_VEL
LIN {X 0,Y 439.363,Z 189.752,A -85,B 0,C 180,E1 -9032.031,E2 -9032.031} C_VEL
LIN {X 0,Y 439.387,Z 189.754,A -85,B 0,C 180,E1 -9035.341,E2 -9035.341} C_VEL
LIN {X 0,Y 439.372,Z 189.753,A -85,B 0,C 180,E1 -9038.597,E2 -9038.597} C_VEL
LIN {X 0,Y 439.384,Z 189.754,A -85,B 0,C 180,E1 -9041.258,E2 -9041.258} C_VEL
LIN {X 0,Y 439.397,Z 189.752,A -85,B 0,C 180,E1 -9044.73,E2 -9044.73} C_VEL
LIN {X 0,Y 439.381,Z 189.75,A -85,B 0,C 180,E1 -9047.795,E2 -9047.795} C_VEL
LIN {X 0,Y 439.391,Z 189.749,A -85,B 0,C 180,E1 -9050.225,E2 -9050.225} C_VEL
LIN {X 0,Y 439.37,Z 189.751,A -85,B 0,C 180,E1 -9053.714,E2 -9053.714} C_VEL
LIN {X 0,Y 439.371,Z 189.758,A -85,B 0,C 180,E1 -9057.055,E2 -9057.055} C_VEL
LIN {X 0,Y 439.377,Z 189.757,A -85,B 0,C 180,E1 -9060.275,E2 -9060.275} C_VEL
LIN {X 0,Y 439.462,Z 189.925,A -85,B 0,C 180,E1 -9061.465,E2 -9061.465} C_VEL
LIN {X 0,Y 443.155,Z 206.39,A -85,B 0,C 180,E1 -9064.145,E2 -9064.145} C_VEL
LIN {X 0,Y 443.541,Z 209.833,A -85,B 0,C 180,E1 -9064.672,E2 -9064.672} C_VEL
LIN {X 0,Y 442.241,Z 231.855,A -85,B 0,C 180,E1 -9067.826,E2 -9067.826} C_VEL
LIN {X 0,Y 440.948,Z 257.178,A -85,B 0,C 180,E1 -9071.412,E2 -9071.412} C_VEL
LIN {X 0,Y 440.616,Z 264.167,A -85,B 0,C 180,E1 -9072.387,E2 -9072.387} C_VEL
LIN {X 0,Y 442.912,Z 286.41,A -85,B 0,C 180,E1 -9072.878,E2 -9072.878} C_VEL
LIN {X 0,Y 442.044,Z 372.379,A -85,B 0,C 180,E1 -9074.379,E2 -9074.379} C_VEL
LIN {X 0,Y 441.617,Z 385.943,A -85,B 0,C 180,E1 -9074.807,E2 -9074.807} C_VEL
LIN {X 0,Y 441.126,Z 398.659,A -85,B 0,C 180,E1 -9075.409,E2 -9075.409} C_VEL
LIN {X 0,Y 440.579,Z 410.343,A -85,B 0,C 180,E1 -9076.157,E2 -9076.157} C_VEL
LIN {X 0,Y 440.052,Z 421.637,A -85,B 0,C 180,E1 -9077.081,E2 -9077.081} C_VEL
LIN {X 0,Y 439.567,Z 430.737,A -85,B 0,C 180,E1 -9078.004,E2 -9078.004} C_VEL
LIN {X 0,Y 439.182,Z 440.049,A -85,B 0,C 180,E1 -9079.163,E2 -9079.163} C_VEL
LIN {X 0,Y 438.795,Z 449.081,A -85,B 0,C 180,E1 -9080.552,E2 -9080.552} C_VEL
LIN {X 0,Y 438.647,Z 456.296,A -85,B 0,C 180,E1 -9081.942,E2 -9081.942} C_VEL
LIN {X 0,Y 438.526,Z 462.83,A -85,B 0,C 180,E1 -9083.559,E2 -9083.559} C_VEL
LIN {X 0,Y 438.464,Z 467.087,A -85,B 0,C 180,E1 -9084.943,E2 -9084.943} C_VEL
LIN {X 0,Y 438.57,Z 470.237,A -85,B 0,C 180,E1 -9086.326,E2 -9086.326} C_VEL
LIN {X 0,Y 438.621,Z 471.777,A -85,B 0,C 180,E1 -9087.245,E2 -9087.245} C_VEL
LIN {X 0,Y 438.499,Z 472.818,A -85,B 0,C 180,E1 -9088.164,E2 -9088.164} C_VEL
LIN {X 0,Y 438.452,Z 473.45,A -85,B 0,C 180,E1 -9089.082,E2 -9089.082} C_VEL
LIN {X 0,Y 438.469,Z 473.68,A -85,B 0,C 180,E1 -9090.001,E2 -9090.001} C_VEL
LIN {X 0,Y 438.454,Z 473.468,A -85,B 0,C 180,E1 -9090.919,E2 -9090.919} C_VEL
LIN {X 0,Y 438.502,Z 472.818,A -85,B 0,C 180,E1 -9091.838,E2 -9091.838} C_VEL
LIN {X 0,Y 438.608,Z 471.764,A -85,B 0,C 180,E1 -9092.756,E2 -9092.756} C_VEL
LIN {X 0,Y 438.581,Z 470.277,A -85,B 0,C 180,E1 -9093.676,E2 -9093.676} C_VEL
LIN {X 0,Y 438.471,Z 467.153,A -85,B 0,C 180,E1 -9095.058,E2 -9095.058} C_VEL
LIN {X 0,Y 438.507,Z 462.942,A -85,B 0,C 180,E1 -9096.442,E2 -9096.442} C_VEL
LIN {X 0,Y 438.648,Z 456.466,A -85,B 0,C 180,E1 -9098.06,E2 -9098.06} C_VEL
LIN {X 0,Y 438.797,Z 449.413,A -85,B 0,C 180,E1 -9099.45,E2 -9099.45} C_VEL
LIN {X 0,Y 439.093,Z 442.222,A -85,B 0,C 180,E1 -9100.607,E2 -9100.607} C_VEL
LIN {X 0,Y 439.463,Z 433.544,A -85,B 0,C 180,E1 -9101.766,E2 -9101.766} C_VEL
LIN {X 0,Y 440.016,Z 423.533,A -85,B 0,C 180,E1 -9102.851,E2 -9102.851} C_VEL
LIN {X 0,Y 440.577,Z 412.174,A -85,B 0,C 180,E1 -9103.844,E2 -9103.844} C_VEL
LIN {X 0,Y 441.261,Z 400.421,A -85,B 0,C 180,E1 -9104.646,E2 -9104.646} C_VEL
LIN {X 0,Y 441.882,Z 386.892,A -85,B 0,C 180,E1 -9105.333,E2 -9105.333} C_VEL
LIN {X 0,Y 442.345,Z 374.848,A -85,B 0,C 180,E1 -9105.759,E2 -9105.759} C_VEL
LIN {X 0,Y 442.628,Z 359.945,A -85,B 0,C 180,E1 -9106.074,E2 -9106.074} C_VEL
LIN {X 0,Y 443.406,Z 284.869,A -85,B 0,C 180,E1 -9107.408,E2 -9107.408} C_VEL
LIN {X 0,Y 440.85,Z 262.922,A -85,B 0,C 180,E1 -9107.956,E2 -9107.956} C_VEL
LIN {X 0,Y 441.671,Z 244.149,A -85,B 0,C 180,E1 -9110.492,E2 -9110.492} C_VEL
LIN {X 0,Y 442.827,Z 221.465,A -85,B 0,C 180,E1 -9113.625,E2 -9113.625} C_VEL
LIN {X 0,Y 443.495,Z 207.551,A -85,B 0,C 180,E1 -9115.583,E2 -9115.583} C_VEL
LIN {X 0,Y 440.807,Z 195.281,A -85,B 0,C 180,E1 -9117.54,E2 -9117.54} C_VEL
LIN {X 0,Y 439.426,Z 189.879,A -85,B 0,C 180,E1 -9118.486,E2 -9118.486} C_VEL
LIN {X 0,Y 439.375,Z 189.756,A -85,B 0,C 180,E1 -9121.861,E2 -9121.861} C_VEL
LIN {X 0,Y 439.399,Z 189.755,A -85,B 0,C 180,E1 -9125.156,E2 -9125.156} C_VEL
LIN {X 0,Y 439.365,Z 189.756,A -85,B 0,C 180,E1 -9128.597,E2 -9128.597} C_VEL
LIN {X 0,Y 439.361,Z 189.755,A -85,B 0,C 180,E1 -9132.209,E2 -9132.209} C_VEL
LIN {X 0,Y 439.401,Z 189.752,A -85,B 0,C 180,E1 -9135.27,E2 -9135.27} C_VEL
LIN {X 0,Y 439.384,Z 189.754,A -85,B 0,C 180,E1 -9138.744,E2 -9138.744} C_VEL
LIN {X 0,Y 439.375,Z 189.752,A -85,B 0,C 180,E1 -9141.608,E2 -9141.608} C_VEL
LIN {X 0,Y 439.399,Z 189.753,A -85,B 0,C 180,E1 -9144.844,E2 -9144.844} C_VEL
LIN {X 0,Y 439.374,Z 189.753,A -85,B 0,C 180,E1 -9148.139,E2 -9148.139} C_VEL
LIN {X 0,Y 439.435,Z 189.745,A -85,B 0,C 180,E1 -9151.598,E2 -9151.598} C_VEL
LIN {X 0,Y 439.4,Z 189.754,A -85,B 0,C 180,E1 -9154.414,E2 -9154.414} C_VEL
LIN {X 0,Y 439.366,Z 189.753,A -85,B 0,C 180,E1 -9157.424,E2 -9157.424} C_VEL
LIN {X 0,Y 439.443,Z 189.747,A -85,B 0,C 180,E1 -9160.663,E2 -9160.663} C_VEL
LIN {X 0,Y 439.464,Z 189.745,A -85,B 0,C 180,E1 -9164.224,E2 -9164.224} C_VEL
LIN {X 0,Y 439.485,Z 189.741,A -85,B 0,C 180,E1 -9168.001,E2 -9168.001} C_VEL
LIN {X 0,Y 439.498,Z 189.741,A -85,B 0,C 180,E1 -9170.798,E2 -9170.798} C_VEL
LIN {X 0,Y 439.591,Z 189.728,A -85,B 0,C 180,E1 -9173.574,E2 -9173.574} C_VEL
LIN {X 0,Y 439.64,Z 189.724,A -85,B 0,C 180,E1 -9177.251,E2 -9177.251} C_VEL
LIN {X 0,Y 439.67,Z 189.938,A -85,B 0,C 180,E1 -9177.996,E2 -9177.996} C_VEL
LIN {X 0,Y 441.088,Z 196.673,A -85,B 0,C 180,E1 -9179.315,E2 -9179.315} C_VEL
LIN {X 0,Y 440.851,Z 213.165,A -85,B 0,C 180,E1 -9182.284,E2 -9182.284} C_VEL
LIN {X 0,Y 440.691,Z 228.598,A -85,B 0,C 180,E1 -9185.06,E2 -9185.06} C_VEL
LIN {X 0,Y 443.406,Z 242.593,A -85,B 0,C 180,E1 -9185.514,E2 -9185.514} C_VEL
LIN {X 0,Y 442.248,Z 311.747,A -85,B 0,C 180,E1 -9186.931,E2 -9186.931} C_VEL
LIN {X 0,Y 442.057,Z 323.763,A -85,B 0,C 180,E1 -9187.364,E2 -9187.364} C_VEL
LIN {X 0,Y 441.695,Z 335.721,A -85,B 0,C 180,E1 -9188.003,E2 -9188.003} C_VEL
LIN {X 0,Y 441.294,Z 346.402,A -85,B 0,C 180,E1 -9188.783,E2 -9188.783} C_VEL
LIN {X 0,Y 440.918,Z 355.519,A -85,B 0,C 180,E1 -9189.634,E2 -9189.634} C_VEL
LIN {X 0,Y 440.47,Z 363.565,A -85,B 0,C 180,E1 -9190.573,E2 -9190.573} C_VEL
LIN {X 0,Y 439.994,Z 371.667,A -85,B 0,C 180,E1 -9191.75,E2 -9191.75} C_VEL
LIN {X 0,Y 439.607,Z 379.164,A -85,B 0,C 180,E1 -9193.168,E2 -9193.168} C_VEL
LIN {X 0,Y 439.294,Z 383.989,A -85,B 0,C 180,E1 -9194.357,E2 -9194.357} C_VEL
LIN {X 0,Y 439.031,Z 388.352,A -85,B 0,C 180,E1 -9195.791,E2 -9195.791} C_VEL
LIN {X 0,Y 438.903,Z 390.445,A -85,B 0,C 180,E1 -9196.751,E2 -9196.751} C_VEL
LIN {X 0,Y 438.78,Z 391.968,A -85,B 0,C 180,E1 -9197.717,E2 -9197.717} C_VEL
LIN {X 0,Y 438.692,Z 393.097,A -85,B 0,C 180,E1 -9199.056,E2 -9199.056} C_VEL
LIN {X 0,Y 438.623,Z 393.055,A -85,B 0,C 180,E1 -9200.64,E2 -9200.64} C_VEL
LIN {X 0,Y 438.642,Z 392.2,A -85,B 0,C 180,E1 -9201.676,E2 -9201.676} C_VEL
LIN {X 0,Y 438.767,Z 389.913,A -85,B 0,C 180,E1 -9203.105,E2 -9203.105} C_VEL
LIN {X 0,Y 438.952,Z 386.122,A -85,B 0,C 180,E1 -9204.6,E2 -9204.6} C_VEL
LIN {X 0,Y 439.145,Z 381.14,A -85,B 0,C 180,E1 -9205.98,E2 -9205.98} C_VEL
LIN {X 0,Y 439.363,Z 375.825,A -85,B 0,C 180,E1 -9207.121,E2 -9207.121} C_VEL
LIN {X 0,Y 439.716,Z 368.35,A -85,B 0,C 180,E1 -9208.383,E2 -9208.383} C_VEL
LIN {X 0,Y 440.073,Z 359.623,A -85,B 0,C 180,E1 -9209.542,E2 -9209.542} C_VEL
LIN {X 0,Y 440.459,Z 349.981,A -85,B 0,C 180,E1 -9210.55,E2 -9210.55} C_VEL
LIN {X 0,Y 440.816,Z 340.286,A -85,B 0,C 180,E1 -9211.341,E2 -9211.341} C_VEL
LIN {X 0,Y 441.126,Z 329.837,A -85,B 0,C 180,E1 -9212.006,E2 -9212.006} C_VEL
LIN {X 0,Y 441.401,Z 317.541,A -85,B 0,C 180,E1 -9212.564,E2 -9212.564} C_VEL
LIN {X 0,Y 441.509,Z 305.952,A -85,B 0,C 180,E1 -9212.902,E2 -9212.902} C_VEL
LIN {X 0,Y 442.241,Z 240.821,A -85,B 0,C 180,E1 -9214.12,E2 -9214.12} C_VEL
LIN {X 0,Y 439.99,Z 227.539,A -85,B 0,C 180,E1 -9214.465,E2 -9214.465} C_VEL
LIN {X 0,Y 440.328,Z 213.151,A -85,B 0,C 180,E1 -9217.337,E2 -9217.337} C_VEL
LIN {X 0,Y 440.655,Z 197.338,A -85,B 0,C 180,E1 -9220.61,E2 -9220.61} C_VEL
LIN {X 0,Y 439.498,Z 190.136,A -85,B 0,C 180,E1 -9222.192,E2 -9222.192} C_VEL
LIN {X 0,Y 439.43,Z 189.752,A -85,B 0,C 180,E1 -9222.413,E2 -9222.413} C_VEL
LIN {X 0,Y 439.398,Z 189.752,A -85,B 0,C 180,E1 -9225.27,E2 -9225.27} C_VEL
LIN {X 0,Y 439.387,Z 189.749,A -85,B 0,C 180,E1 -9228.743,E2 -9228.743} C_VEL
LIN {X 0,Y 439.37,Z 189.758,A -85,B 0,C 180,E1 -9231.608,E2 -9231.608} C_VEL
LIN {X 0,Y 439.399,Z 189.747,A -85,B 0,C 180,E1 -9234.844,E2 -9234.844} C_VEL
LIN {X 0,Y 439.371,Z 189.752,A -85,B 0,C 180,E1 -9238.139,E2 -9238.139} C_VEL
LIN {X 0,Y 439.428,Z 189.749,A -85,B 0,C 180,E1 -9241.692,E2 -9241.692} C_VEL
LIN {X 0,Y 438.758,Z 189.827,A -85,B 0,C 180,E1 -9242.456,E2 -9242.456} C_VEL
LIN {X 0,Y 435.912,Z 190.187,A -85,B 0,C 180,E1 -9243.698,E2 -9243.698} C_VEL
LIN {X 0,Y 433.502,Z 190.491,A -85,B 0,C 180,E1 -9244.701,E2 -9244.701} C_VEL
LIN {X 0,Y 432.461,Z 190.619,A -85,B 0,C 180,E1 -9245.475,E2 -9245.475} C_VEL
LIN {X 0,Y 432.373,Z 190.627,A -85,B 0,C 180,E1 -9245.737,E2 -9245.737} C_VEL
LIN {X 0,Y 432.349,Z 190.629,A -85,B 0,C 180,E1 -9249.046,E2 -9249.046} C_VEL
LIN {X 0,Y 432.376,Z 190.623,A -85,B 0,C 180,E1 -9252.011,E2 -9252.011} C_VEL
LIN {X 0,Y 432.395,Z 190.623,A -85,B 0,C 180,E1 -9254.926,E2 -9254.926} C_VEL
LIN {X 0,Y 432.457,Z 190.614,A -85,B 0,C 180,E1 -9257.803,E2 -9257.803} C_VEL
LIN {X 0,Y 432.49,Z 190.611,A -85,B 0,C 180,E1 -9261.59,E2 -9261.59} C_VEL
LIN {X 0,Y 432.597,Z 190.595,A -85,B 0,C 180,E1 -9264.406,E2 -9264.406} C_VEL
LIN {X 0,Y 432.603,Z 190.594,A -85,B 0,C 180,E1 -9268.137,E2 -9268.137} C_VEL
LIN {X 0,Y 432.731,Z 190.578,A -85,B 0,C 180,E1 -9269.999,E2 -9269.999} C_VEL
LIN {X 0,Y 432.602,Z 190.598,A -85,B 0,C 180,E1 -9272.793,E2 -9272.793} C_VEL
LIN {X 0,Y 432.561,Z 190.601,A -85,B 0,C 180,E1 -9276.53,E2 -9276.53} C_VEL
LIN {X 0,Y 432.439,Z 190.617,A -85,B 0,C 180,E1 -9279.352,E2 -9279.352} C_VEL
LIN {X 0,Y 432.427,Z 190.622,A -85,B 0,C 180,E1 -9282.803,E2 -9282.803} C_VEL
LIN {X 0,Y 432.408,Z 190.621,A -85,B 0,C 180,E1 -9286.478,E2 -9286.478} C_VEL
LIN {X 0,Y 432.334,Z 190.628,A -85,B 0,C 180,E1 -9289.96,E2 -9289.96} C_VEL
LIN {X 0,Y 432.314,Z 190.634,A -85,B 0,C 180,E1 -9292.964,E2 -9292.964} C_VEL
LIN {X 0,Y 432.359,Z 190.625,A -85,B 0,C 180,E1 -9296.032,E2 -9296.032} C_VEL
LIN {X 0,Y 432.337,Z 190.628,A -85,B 0,C 180,E1 -9299.187,E2 -9299.187} C_VEL
LIN {X 0,Y 432.317,Z 190.635,A -85,B 0,C 180,E1 -9302.442,E2 -9302.442} C_VEL
LIN {X 0,Y 432.342,Z 190.626,A -85,B 0,C 180,E1 -9305.632,E2 -9305.632} C_VEL
LIN {X 0,Y 432.358,Z 190.624,A -85,B 0,C 180,E1 -9309.341,E2 -9309.341} C_VEL
LIN {X 0,Y 432.366,Z 190.624,A -85,B 0,C 180,E1 -9311.792,E2 -9311.792} C_VEL
LIN {X 0,Y 432.37,Z 190.63,A -85,B 0,C 180,E1 -9314.341,E2 -9314.341} C_VEL
LIN {X 0,Y 432.358,Z 190.631,A -85,B 0,C 180,E1 -9318.393,E2 -9318.393} C_VEL
LIN {X 0,Y 432.343,Z 190.629,A -85,B 0,C 180,E1 -9321.851,E2 -9321.851} C_VEL
LIN {X 0,Y 432.332,Z 190.628,A -85,B 0,C 180,E1 -9325.323,E2 -9325.323} C_VEL
LIN {X 0,Y 432.324,Z 190.631,A -85,B 0,C 180,E1 -9328.655,E2 -9328.655} C_VEL
LIN {X 0,Y 432.375,Z 190.627,A -85,B 0,C 180,E1 -9331.877,E2 -9331.877} C_VEL
LIN {X 0,Y 432.343,Z 190.626,A -85,B 0,C 180,E1 -9334.999,E2 -9334.999} C_VEL
LIN {X 0,Y 432.349,Z 190.633,A -85,B 0,C 180,E1 -9338.046,E2 -9338.046} C_VEL
LIN {X 0,Y 432.378,Z 190.622,A -85,B 0,C 180,E1 -9341.03,E2 -9341.03} C_VEL
LIN {X 0,Y 432.434,Z 190.622,A -85,B 0,C 180,E1 -9343.962,E2 -9343.962} C_VEL
LIN {X 0,Y 432.451,Z 190.62,A -85,B 0,C 180,E1 -9347.804,E2 -9347.804} C_VEL
LIN {X 0,Y 432.483,Z 190.614,A -85,B 0,C 180,E1 -9351.591,E2 -9351.591} C_VEL
LIN {X 0,Y 432.589,Z 190.597,A -85,B 0,C 180,E1 -9354.406,E2 -9354.406} C_VEL
LIN {X 0,Y 432.595,Z 190.597,A -85,B 0,C 180,E1 -9358.138,E2 -9358.138} C_VEL
LIN {X 0,Y 432.725,Z 190.582,A -85,B 0,C 180,E1 -9360,E2 -9360} C_VEL
LIN {X 0,Y 432.584,Z 190.596,A -85,B 0,C 180,E1 -9362.794,E2 -9362.794} C_VEL
LIN {X 0,Y 432.56,Z 190.599,A -85,B 0,C 180,E1 -9366.531,E2 -9366.531} C_VEL
LIN {X 0,Y 432.434,Z 190.62,A -85,B 0,C 180,E1 -9369.354,E2 -9369.354} C_VEL
LIN {X 0,Y 432.423,Z 190.617,A -85,B 0,C 180,E1 -9372.804,E2 -9372.804} C_VEL
LIN {X 0,Y 432.405,Z 190.618,A -85,B 0,C 180,E1 -9376.48,E2 -9376.48} C_VEL
LIN {X 0,Y 432.331,Z 190.629,A -85,B 0,C 180,E1 -9379.961,E2 -9379.961} C_VEL
LIN {X 0,Y 432.312,Z 190.633,A -85,B 0,C 180,E1 -9382.965,E2 -9382.965} C_VEL
LIN {X 0,Y 432.358,Z 190.625,A -85,B 0,C 180,E1 -9386.033,E2 -9386.033} C_VEL
LIN {X 0,Y 432.336,Z 190.634,A -85,B 0,C 180,E1 -9389.188,E2 -9389.188} C_VEL
LIN {X 0,Y 432.317,Z 190.63,A -85,B 0,C 180,E1 -9392.444,E2 -9392.444} C_VEL
LIN {X 0,Y 432.338,Z 190.629,A -85,B 0,C 180,E1 -9395.632,E2 -9395.632} C_VEL
LIN {X 0,Y 432.336,Z 190.63,A -85,B 0,C 180,E1 -9398.715,E2 -9398.715} C_VEL
LIN {X 0,Y 432.329,Z 190.628,A -85,B 0,C 180,E1 -9401.798,E2 -9401.798} C_VEL
LIN {X 0,Y 432.33,Z 190.629,A -85,B 0,C 180,E1 -9404.348,E2 -9404.348} C_VEL
LIN {X 0,Y 432.313,Z 190.637,A -85,B 0,C 180,E1 -9407.017,E2 -9407.017} C_VEL
LIN {X 0,Y 432.329,Z 190.628,A -85,B 0,C 180,E1 -9409.822,E2 -9409.822} C_VEL
LIN {X 0,Y 432.302,Z 190.638,A -85,B 0,C 180,E1 -9413.023,E2 -9413.023} C_VEL
LIN {X 0,Y 432.357,Z 190.628,A -85,B 0,C 180,E1 -9415.998,E2 -9415.998} C_VEL
LIN {X 0,Y 432.345,Z 190.632,A -85,B 0,C 180,E1 -9419.491,E2 -9419.491} C_VEL
LIN {X 0,Y 432.402,Z 190.802,A -85,B 0,C 180,E1 -9421.203,E2 -9421.203} C_VEL
LIN {X 0,Y 435.753,Z 205.653,A -85,B 0,C 180,E1 -9423.672,E2 -9423.672} C_VEL
LIN {X 0,Y 436.664,Z 210.92,A -85,B 0,C 180,E1 -9424.508,E2 -9424.508} C_VEL
LIN {X 0,Y 435.294,Z 232.865,A -85,B 0,C 180,E1 -9427.703,E2 -9427.703} C_VEL
LIN {X 0,Y 434.001,Z 256.47,A -85,B 0,C 180,E1 -9431.104,E2 -9431.104} C_VEL
LIN {X 0,Y 433.65,Z 264.046,A -85,B 0,C 180,E1 -9432.169,E2 -9432.169} C_VEL
LIN {X 0,Y 435.997,Z 286.785,A -85,B 0,C 180,E1 -9432.673,E2 -9432.673} C_VEL
LIN {X 0,Y 435.117,Z 371.809,A -85,B 0,C 180,E1 -9434.184,E2 -9434.184} C_VEL
LIN {X 0,Y 434.707,Z 384.627,A -85,B 0,C 180,E1 -9434.589,E2 -9434.589} C_VEL
LIN {X 0,Y 434.178,Z 397.096,A -85,B 0,C 180,E1 -9435.171,E2 -9435.171} C_VEL
LIN {X 0,Y 433.599,Z 408.996,A -85,B 0,C 180,E1 -9435.93,E2 -9435.93} C_VEL
LIN {X 0,Y 433.047,Z 420.441,A -85,B 0,C 180,E1 -9436.868,E2 -9436.868} C_VEL
LIN {X 0,Y 432.605,Z 429.675,A -85,B 0,C 180,E1 -9437.808,E2 -9437.808} C_VEL
LIN {X 0,Y 432.132,Z 439.089,A -85,B 0,C 180,E1 -9438.984,E2 -9438.984} C_VEL
LIN {X 0,Y 431.736,Z 448.188,A -85,B 0,C 180,E1 -9440.396,E2 -9440.396} C_VEL
LIN {X 0,Y 431.572,Z 455.474,A -85,B 0,C 180,E1 -9441.809,E2 -9441.809} C_VEL
LIN {X 0,Y 431.463,Z 462.052,A -85,B 0,C 180,E1 -9443.454,E2 -9443.454} C_VEL
LIN {X 0,Y 431.403,Z 466.345,A -85,B 0,C 180,E1 -9444.86,E2 -9444.86} C_VEL
LIN {X 0,Y 431.499,Z 469.522,A -85,B 0,C 180,E1 -9446.265,E2 -9446.265} C_VEL
LIN {X 0,Y 431.568,Z 471.081,A -85,B 0,C 180,E1 -9447.2,E2 -9447.2} C_VEL
LIN {X 0,Y 431.444,Z 472.141,A -85,B 0,C 180,E1 -9448.134,E2 -9448.134} C_VEL
LIN {X 0,Y 431.389,Z 472.78,A -85,B 0,C 180,E1 -9449.067,E2 -9449.067} C_VEL
LIN {X 0,Y 431.401,Z 473.017,A -85,B 0,C 180,E1 -9450.001,E2 -9450.001} C_VEL
LIN {X 0,Y 431.39,Z 472.821,A -85,B 0,C 180,E1 -9450.934,E2 -9450.934} C_VEL
LIN {X 0,Y 431.447,Z 472.175,A -85,B 0,C 180,E1 -9451.868,E2 -9451.868} C_VEL
LIN {X 0,Y 431.526,Z 471.122,A -85,B 0,C 180,E1 -9452.801,E2 -9452.801} C_VEL
LIN {X 0,Y 431.49,Z 469.641,A -85,B 0,C 180,E1 -9453.736,E2 -9453.736} C_VEL
LIN {X 0,Y 431.405,Z 466.527,A -85,B 0,C 180,E1 -9455.141,E2 -9455.141} C_VEL
LIN {X 0,Y 431.443,Z 462.326,A -85,B 0,C 180,E1 -9456.548,E2 -9456.548} C_VEL
LIN {X 0,Y 431.573,Z 455.856,A -85,B 0,C 180,E1 -9458.193,E2 -9458.193} C_VEL
LIN {X 0,Y 431.751,Z 448.804,A -85,B 0,C 180,E1 -9459.605,E2 -9459.605} C_VEL
LIN {X 0,Y 432.072,Z 441.626,A -85,B 0,C 180,E1 -9460.782,E2 -9460.782} C_VEL
LIN {X 0,Y 432.448,Z 432.967,A -85,B 0,C 180,E1 -9461.959,E2 -9461.959} C_VEL
LIN {X 0,Y 432.99,Z 424.054,A -85,B 0,C 180,E1 -9462.956,E2 -9462.956} C_VEL
LIN {X 0,Y 433.547,Z 413.235,A -85,B 0,C 180,E1 -9463.942,E2 -9463.942} C_VEL
LIN {X 0,Y 434.272,Z 401.78,A -85,B 0,C 180,E1 -9464.768,E2 -9464.768} C_VEL
LIN {X 0,Y 434.918,Z 389.06,A -85,B 0,C 180,E1 -9465.464,E2 -9465.464} C_VEL
LIN {X 0,Y 435.479,Z 375.466,A -85,B 0,C 180,E1 -9465.984,E2 -9465.984} C_VEL
LIN {X 0,Y 435.807,Z 361.668,A -85,B 0,C 180,E1 -9466.302,E2 -9466.302} C_VEL
LIN {X 0,Y 436.629,Z 285.199,A -85,B 0,C 180,E1 -9467.696,E2 -9467.696} C_VEL
LIN {X 0,Y 434.036,Z 262.801,A -85,B 0,C 180,E1 -9468.267,E2 -9468.267} C_VEL
LIN {X 0,Y 434.087,Z 259.809,A -85,B 0,C 180,E1 -9468.624,E2 -9468.624} C_VEL
LIN {X 0,Y 435.393,Z 233.525,A -85,B 0,C 180,E1 -9472.293,E2 -9472.293} C_VEL
LIN {X 0,Y 436.737,Z 210.981,A -85,B 0,C 180,E1 -9475.491,E2 -9475.491} C_VEL
LIN {X 0,Y 436.347,Z 207.441,A -85,B 0,C 180,E1 -9476.034,E2 -9476.034} C_VEL
LIN {X 0,Y 433.573,Z 195.304,A -85,B 0,C 180,E1 -9478.04,E2 -9478.04} C_VEL
LIN {X 0,Y 432.4,Z 190.755,A -85,B 0,C 180,E1 -9478.861,E2 -9478.861} C_VEL
LIN {X 0,Y 432.328,Z 190.634,A -85,B 0,C 180,E1 -9482.293,E2 -9482.293} C_VEL
LIN {X 0,Y 432.34,Z 190.633,A -85,B 0,C 180,E1 -9484.677,E2 -9484.677} C_VEL
LIN {X 0,Y 432.332,Z 190.63,A -85,B 0,C 180,E1 -9488.151,E2 -9488.151} C_VEL
LIN {X 0,Y 432.312,Z 190.634,A -85,B 0,C 180,E1 -9491.8,E2 -9491.8} C_VEL
LIN {X 0,Y 432.336,Z 190.63,A -85,B 0,C 180,E1 -9494.347,E2 -9494.347} C_VEL
LIN {X 0,Y 432.319,Z 190.637,A -85,B 0,C 180,E1 -9497.016,E2 -9497.016} C_VEL
LIN {X 0,Y 432.334,Z 190.628,A -85,B 0,C 180,E1 -9499.821,E2 -9499.821} C_VEL
LIN {X 0,Y 432.309,Z 190.637,A -85,B 0,C 180,E1 -9503.022,E2 -9503.022} C_VEL
LIN {X 0,Y 432.36,Z 190.626,A -85,B 0,C 180,E1 -9505.997,E2 -9505.997} C_VEL
LIN {X 0,Y 432.349,Z 190.628,A -85,B 0,C 180,E1 -9509.49,E2 -9509.49} C_VEL
LIN {X 0,Y 432.393,Z 190.624,A -85,B 0,C 180,E1 -9512.928,E2 -9512.928} C_VEL
LIN {X 0,Y 432.37,Z 190.626,A -85,B 0,C 180,E1 -9516.023,E2 -9516.023} C_VEL
LIN {X 0,Y 432.352,Z 190.628,A -85,B 0,C 180,E1 -9519.046,E2 -9519.046} C_VEL
LIN {X 0,Y 432.374,Z 190.627,A -85,B 0,C 180,E1 -9522.011,E2 -9522.011} C_VEL
LIN {X 0,Y 432.396,Z 190.625,A -85,B 0,C 180,E1 -9524.926,E2 -9524.926} C_VEL
LIN {X 0,Y 432.461,Z 190.615,A -85,B 0,C 180,E1 -9527.803,E2 -9527.803} C_VEL
LIN {X 0,Y 432.465,Z 190.615,A -85,B 0,C 180,E1 -9531.589,E2 -9531.589} C_VEL
LIN {X 0,Y 432.585,Z 190.604,A -85,B 0,C 180,E1 -9534.406,E2 -9534.406} C_VEL
LIN {X 0,Y 432.607,Z 190.779,A -85,B 0,C 180,E1 -9537.643,E2 -9537.643} C_VEL
LIN {X 0,Y 434.284,Z 199.106,A -85,B 0,C 180,E1 -9539.304,E2 -9539.304} C_VEL
LIN {X 0,Y 433.96,Z 215.668,A -85,B 0,C 180,E1 -9542.32,E2 -9542.32} C_VEL
LIN {X 0,Y 433.844,Z 229.028,A -85,B 0,C 180,E1 -9544.733,E2 -9544.733} C_VEL
LIN {X 0,Y 436.63,Z 242.614,A -85,B 0,C 180,E1 -9545.194,E2 -9545.194} C_VEL
LIN {X 0,Y 435.448,Z 312.821,A -85,B 0,C 180,E1 -9546.69,E2 -9546.69} C_VEL
LIN {X 0,Y 435.241,Z 324.635,A -85,B 0,C 180,E1 -9547.13,E2 -9547.13} C_VEL
LIN {X 0,Y 434.856,Z 336.519,A -85,B 0,C 180,E1 -9547.779,E2 -9547.779} C_VEL
LIN {X 0,Y 434.401,Z 348.07,A -85,B 0,C 180,E1 -9548.648,E2 -9548.648} C_VEL
LIN {X 0,Y 433.915,Z 357.362,A -85,B 0,C 180,E1 -9549.556,E2 -9549.556} C_VEL
LIN {X 0,Y 433.504,Z 365.195,A -85,B 0,C 180,E1 -9550.508,E2 -9550.508} C_VEL
LIN {X 0,Y 433.013,Z 373.073,A -85,B 0,C 180,E1 -9551.705,E2 -9551.705} C_VEL
LIN {X 0,Y 432.651,Z 379.435,A -85,B 0,C 180,E1 -9552.93,E2 -9552.93} C_VEL
LIN {X 0,Y 432.322,Z 384.278,A -85,B 0,C 180,E1 -9554.113,E2 -9554.113} C_VEL
LIN {X 0,Y 432.038,Z 388.722,A -85,B 0,C 180,E1 -9555.569,E2 -9555.569} C_VEL
LIN {X 0,Y 431.83,Z 391.77,A -85,B 0,C 180,E1 -9557.034,E2 -9557.034} C_VEL
LIN {X 0,Y 431.682,Z 393.064,A -85,B 0,C 180,E1 -9558.018,E2 -9558.018} C_VEL
LIN {X 0,Y 431.624,Z 393.844,A -85,B 0,C 180,E1 -9559.196,E2 -9559.196} C_VEL
LIN {X 0,Y 431.575,Z 393.923,A -85,B 0,C 180,E1 -9559.997,E2 -9559.997} C_VEL
LIN {X 0,Y 431.554,Z 393.478,A -85,B 0,C 180,E1 -9560.994,E2 -9560.994} C_VEL
LIN {X 0,Y 431.594,Z 392.443,A -85,B 0,C 180,E1 -9561.995,E2 -9561.995} C_VEL
LIN {X 0,Y 431.759,Z 389.763,A -85,B 0,C 180,E1 -9563.503,E2 -9563.503} C_VEL
LIN {X 0,Y 431.962,Z 385.528,A -85,B 0,C 180,E1 -9565.025,E2 -9565.025} C_VEL
LIN {X 0,Y 432.184,Z 379.491,A -85,B 0,C 180,E1 -9566.57,E2 -9566.57} C_VEL
LIN {X 0,Y 432.476,Z 372.89,A -85,B 0,C 180,E1 -9567.852,E2 -9567.852} C_VEL
LIN {X 0,Y 432.886,Z 364.33,A -85,B 0,C 180,E1 -9569.147,E2 -9569.147} C_VEL
LIN {X 0,Y 433.286,Z 355.554,A -85,B 0,C 180,E1 -9570.187,E2 -9570.187} C_VEL
LIN {X 0,Y 433.688,Z 345.978,A -85,B 0,C 180,E1 -9571.091,E2 -9571.091} C_VEL
LIN {X 0,Y 434.052,Z 335.108,A -85,B 0,C 180,E1 -9571.887,E2 -9571.887} C_VEL
LIN {X 0,Y 434.393,Z 323.433,A -85,B 0,C 180,E1 -9572.514,E2 -9572.514} C_VEL
LIN {X 0,Y 434.538,Z 312.069,A -85,B 0,C 180,E1 -9572.939,E2 -9572.939} C_VEL
LIN {X 0,Y 434.72,Z 292.911,A -85,B 0,C 180,E1 -9573.344,E2 -9573.344} C_VEL
LIN {X 0,Y 435.302,Z 241.512,A -85,B 0,C 180,E1 -9574.324,E2 -9574.324} C_VEL
LIN {X 0,Y 433.004,Z 227.726,A -85,B 0,C 180,E1 -9574.695,E2 -9574.695} C_VEL
LIN {X 0,Y 433.372,Z 213.229,A -85,B 0,C 180,E1 -9577.619,E2 -9577.619} C_VEL
LIN {X 0,Y 433.694,Z 198.445,A -85,B 0,C 180,E1 -9580.711,E2 -9580.711} C_VEL
LIN {X 0,Y 432.393,Z 190.719,A -85,B 0,C 180,E1 -9582.469,E2 -9582.469} C_VEL
LIN {X 0,Y 432.332,Z 190.635,A -85,B 0,C 180,E1 -9585.664,E2 -9585.664} C_VEL
LIN {X 0,Y 432.331,Z 190.63,A -85,B 0,C 180,E1 -9588.398,E2 -9588.398} C_VEL
LIN {X 0,Y 432.334,Z 190.633,A -85,B 0,C 180,E1 -9591.849,E2 -9591.849} C_VEL
LIN {X 0,Y 432.339,Z 190.63,A -85,B 0,C 180,E1 -9595.323,E2 -9595.323} C_VEL
LIN {X 0,Y 432.319,Z 190.629,A -85,B 0,C 180,E1 -9598.653,E2 -9598.653} C_VEL
LIN {X 0,Y 432.381,Z 190.625,A -85,B 0,C 180,E1 -9601.876,E2 -9601.876} C_VEL
LIN {X 0,Y 432.35,Z 190.627,A -85,B 0,C 180,E1 -9604.998,E2 -9604.998} C_VEL
LIN {X 0,Y 432.373,Z 190.627,A -85,B 0,C 180,E1 -9605.737,E2 -9605.737} C_VEL
LIN {X 0,Y 431.69,Z 190.708,A -85,B 0,C 180,E1 -9606.514,E2 -9606.514} C_VEL
LIN {X 0,Y 428.812,Z 191.069,A -85,B 0,C 180,E1 -9607.776,E2 -9607.776} C_VEL
LIN {X 0,Y 426.394,Z 191.374,A -85,B 0,C 180,E1 -9608.795,E2 -9608.795} C_VEL
LIN {X 0,Y 425.371,Z 191.5,A -85,B 0,C 180,E1 -9609.583,E2 -9609.583} C_VEL
LIN {X 0,Y 425.296,Z 191.506,A -85,B 0,C 180,E1 -9609.849,E2 -9609.849} C_VEL
LIN {X 0,Y 425.34,Z 191.499,A -85,B 0,C 180,E1 -9612.697,E2 -9612.697} C_VEL
LIN {X 0,Y 425.347,Z 191.501,A -85,B 0,C 180,E1 -9615.649,E2 -9615.649} C_VEL
LIN {X 0,Y 425.35,Z 191.498,A -85,B 0,C 180,E1 -9618.563,E2 -9618.563} C_VEL
LIN {X 0,Y 425.536,Z 191.475,A -85,B 0,C 180,E1 -9622.407,E2 -9622.407} C_VEL
LIN {X 0,Y 425.553,Z 191.472,A -85,B 0,C 180,E1 -9624.313,E2 -9624.313} C_VEL
LIN {X 0,Y 425.573,Z 191.47,A -85,B 0,C 180,E1 -9628.107,E2 -9628.107} C_VEL
LIN {X 0,Y 425.701,Z 191.454,A -85,B 0,C 180,E1 -9629.999,E2 -9629.999} C_VEL
LIN {X 0,Y 425.554,Z 191.477,A -85,B 0,C 180,E1 -9632.839,E2 -9632.839} C_VEL
LIN {X 0,Y 425.52,Z 191.48,A -85,B 0,C 180,E1 -9636.638,E2 -9636.638} C_VEL
LIN {X 0,Y 425.398,Z 191.493,A -85,B 0,C 180,E1 -9639.509,E2 -9639.509} C_VEL
LIN {X 0,Y 425.389,Z 191.5,A -85,B 0,C 180,E1 -9642.903,E2 -9642.903} C_VEL
LIN {X 0,Y 425.357,Z 191.501,A -85,B 0,C 180,E1 -9646.604,E2 -9646.604} C_VEL
LIN {X 0,Y 425.324,Z 191.501,A -85,B 0,C 180,E1 -9649.635,E2 -9649.635} C_VEL
LIN {X 0,Y 425.302,Z 191.504,A -85,B 0,C 180,E1 -9653.364,E2 -9653.364} C_VEL
LIN {X 0,Y 425.345,Z 191.503,A -85,B 0,C 180,E1 -9656.844,E2 -9656.844} C_VEL
LIN {X 0,Y 425.285,Z 191.505,A -85,B 0,C 180,E1 -9659.719,E2 -9659.719} C_VEL
LIN {X 0,Y 425.276,Z 191.509,A -85,B 0,C 180,E1 -9663.047,E2 -9663.047} C_VEL
LIN {X 0,Y 425.28,Z 191.507,A -85,B 0,C 180,E1 -9665.929,E2 -9665.929} C_VEL
LIN {X 0,Y 425.303,Z 191.505,A -85,B 0,C 180,E1 -9669.045,E2 -9669.045} C_VEL
LIN {X 0,Y 425.324,Z 191.505,A -85,B 0,C 180,E1 -9672.645,E2 -9672.645} C_VEL
LIN {X 0,Y 425.286,Z 191.505,A -85,B 0,C 180,E1 -9675.281,E2 -9675.281} C_VEL
LIN {X 0,Y 425.296,Z 191.508,A -85,B 0,C 180,E1 -9678.625,E2 -9678.625} C_VEL
LIN {X 0,Y 425.313,Z 191.502,A -85,B 0,C 180,E1 -9681.104,E2 -9681.104} C_VEL
LIN {X 0,Y 425.292,Z 191.507,A -85,B 0,C 180,E1 -9684.664,E2 -9684.664} C_VEL
LIN {X 0,Y 425.265,Z 191.514,A -85,B 0,C 180,E1 -9688.074,E2 -9688.074} C_VEL
LIN {X 0,Y 425.329,Z 191.5,A -85,B 0,C 180,E1 -9691.368,E2 -9691.368} C_VEL
LIN {X 0,Y 425.287,Z 191.507,A -85,B 0,C 180,E1 -9694.555,E2 -9694.555} C_VEL
LIN {X 0,Y 425.279,Z 191.509,A -85,B 0,C 180,E1 -9697.661,E2 -9697.661} C_VEL
LIN {X 0,Y 425.353,Z 191.497,A -85,B 0,C 180,E1 -9700.704,E2 -9700.704} C_VEL
LIN {X 0,Y 425.39,Z 191.497,A -85,B 0,C 180,E1 -9703.689,E2 -9703.689} C_VEL
LIN {X 0,Y 425.404,Z 191.495,A -85,B 0,C 180,E1 -9707.598,E2 -9707.598} C_VEL
LIN {X 0,Y 425.434,Z 191.49,A -85,B 0,C 180,E1 -9711.45,E2 -9711.45} C_VEL
LIN {X 0,Y 425.545,Z 191.475,A -85,B 0,C 180,E1 -9714.314,E2 -9714.314} C_VEL
LIN {X 0,Y 425.564,Z 191.473,A -85,B 0,C 180,E1 -9718.108,E2 -9718.108} C_VEL
LIN {X 0,Y 425.694,Z 191.458,A -85,B 0,C 180,E1 -9720,E2 -9720} C_VEL
LIN {X 0,Y 425.538,Z 191.474,A -85,B 0,C 180,E1 -9722.84,E2 -9722.84} C_VEL
LIN {X 0,Y 425.519,Z 191.476,A -85,B 0,C 180,E1 -9726.639,E2 -9726.639} C_VEL
LIN {X 0,Y 425.392,Z 191.5,A -85,B 0,C 180,E1 -9729.51,E2 -9729.51} C_VEL
LIN {X 0,Y 425.386,Z 191.494,A -85,B 0,C 180,E1 -9732.904,E2 -9732.904} C_VEL
LIN {X 0,Y 425.354,Z 191.497,A -85,B 0,C 180,E1 -9736.606,E2 -9736.606} C_VEL
LIN {X 0,Y 425.322,Z 191.505,A -85,B 0,C 180,E1 -9739.636,E2 -9739.636} C_VEL
LIN {X 0,Y 425.3,Z 191.511,A -85,B 0,C 180,E1 -9743.366,E2 -9743.366} C_VEL
LIN {X 0,Y 425.341,Z 191.501,A -85,B 0,C 180,E1 -9746.845,E2 -9746.845} C_VEL
LIN {X 0,Y 425.285,Z 191.507,A -85,B 0,C 180,E1 -9749.72,E2 -9749.72} C_VEL
LIN {X 0,Y 425.276,Z 191.513,A -85,B 0,C 180,E1 -9753.049,E2 -9753.049} C_VEL
LIN {X 0,Y 425.276,Z 191.507,A -85,B 0,C 180,E1 -9755.929,E2 -9755.929} C_VEL
LIN {X 0,Y 425.283,Z 191.513,A -85,B 0,C 180,E1 -9759.043,E2 -9759.043} C_VEL
LIN {X 0,Y 425.286,Z 191.505,A -85,B 0,C 180,E1 -9761.959,E2 -9761.959} C_VEL
LIN {X 0,Y 425.281,Z 191.51,A -85,B 0,C 180,E1 -9765.284,E2 -9765.284} C_VEL
LIN {X 0,Y 425.264,Z 191.512,A -85,B 0,C 180,E1 -9768.622,E2 -9768.622} C_VEL
LIN {X 0,Y 425.294,Z 191.509,A -85,B 0,C 180,E1 -9771.102,E2 -9771.102} C_VEL
LIN {X 0,Y 425.296,Z 191.51,A -85,B 0,C 180,E1 -9774.665,E2 -9774.665} C_VEL
LIN {X 0,Y 425.263,Z 191.513,A -85,B 0,C 180,E1 -9778.074,E2 -9778.074} C_VEL
LIN {X 0,Y 425.354,Z 191.672,A -85,B 0,C 180,E1 -9780.93,E2 -9780.93} C_VEL
LIN {X 0,Y 428.744,Z 206.634,A -85,B 0,C 180,E1 -9783.47,E2 -9783.47} C_VEL
LIN {X 0,Y 429.749,Z 211.789,A -85,B 0,C 180,E1 -9784.309,E2 -9784.309} C_VEL
LIN {X 0,Y 428.45,Z 232.169,A -85,B 0,C 180,E1 -9787.328,E2 -9787.328} C_VEL
LIN {X 0,Y 426.997,Z 257.407,A -85,B 0,C 180,E1 -9791.031,E2 -9791.031} C_VEL
LIN {X 0,Y 426.694,Z 263.876,A -85,B 0,C 180,E1 -9791.937,E2 -9791.937} C_VEL
LIN {X 0,Y 429.081,Z 287.288,A -85,B 0,C 180,E1 -9792.466,E2 -9792.466} C_VEL
LIN {X 0,Y 428.187,Z 371.093,A -85,B 0,C 180,E1 -9793.982,E2 -9793.982} C_VEL
LIN {X 0,Y 427.755,Z 383.962,A -85,B 0,C 180,E1 -9794.394,E2 -9794.394} C_VEL
LIN {X 0,Y 427.23,Z 396.475,A -85,B 0,C 180,E1 -9794.985,E2 -9794.985} C_VEL
LIN {X 0,Y 426.678,Z 407.596,A -85,B 0,C 180,E1 -9795.697,E2 -9795.697} C_VEL
LIN {X 0,Y 426.06,Z 419.186,A -85,B 0,C 180,E1 -9796.649,E2 -9796.649} C_VEL
LIN {X 0,Y 425.553,Z 429.611,A -85,B 0,C 180,E1 -9797.724,E2 -9797.724} C_VEL
LIN {X 0,Y 425.103,Z 438.084,A -85,B 0,C 180,E1 -9798.8,E2 -9798.8} C_VEL
LIN {X 0,Y 424.659,Z 447.25,A -85,B 0,C 180,E1 -9800.234,E2 -9800.234} C_VEL
LIN {X 0,Y 424.491,Z 454.613,A -85,B 0,C 180,E1 -9801.671,E2 -9801.671} C_VEL
LIN {X 0,Y 424.393,Z 459.545,A -85,B 0,C 180,E1 -9802.866,E2 -9802.866} C_VEL
LIN {X 0,Y 424.349,Z 464.294,A -85,B 0,C 180,E1 -9804.298,E2 -9804.298} C_VEL
LIN {X 0,Y 424.321,Z 467.86,A -85,B 0,C 180,E1 -9805.726,E2 -9805.726} C_VEL
LIN {X 0,Y 424.498,Z 470.371,A -85,B 0,C 180,E1 -9807.154,E2 -9807.154} C_VEL
LIN {X 0,Y 424.391,Z 471.456,A -85,B 0,C 180,E1 -9808.103,E2 -9808.103} C_VEL
LIN {X 0,Y 424.327,Z 472.106,A -85,B 0,C 180,E1 -9809.052,E2 -9809.052} C_VEL
LIN {X 0,Y 424.335,Z 472.351,A -85,B 0,C 180,E1 -9810.001,E2 -9810.001} C_VEL
LIN {X 0,Y 424.329,Z 472.172,A -85,B 0,C 180,E1 -9810.95,E2 -9810.95} C_VEL
LIN {X 0,Y 424.393,Z 471.537,A -85,B 0,C 180,E1 -9811.899,E2 -9811.899} C_VEL
LIN {X 0,Y 424.446,Z 470.486,A -85,B 0,C 180,E1 -9812.848,E2 -9812.848} C_VEL
LIN {X 0,Y 424.404,Z 469.01,A -85,B 0,C 180,E1 -9813.799,E2 -9813.799} C_VEL
LIN {X 0,Y 424.338,Z 465.906,A -85,B 0,C 180,E1 -9815.227,E2 -9815.227} C_VEL
LIN {X 0,Y 424.389,Z 461.718,A -85,B 0,C 180,E1 -9816.657,E2 -9816.657} C_VEL
LIN {X 0,Y 424.491,Z 455.263,A -85,B 0,C 180,E1 -9818.33,E2 -9818.33} C_VEL
LIN {X 0,Y 424.7,Z 448.227,A -85,B 0,C 180,E1 -9819.766,E2 -9819.766} C_VEL
LIN {X 0,Y 425.058,Z 441.058,A -85,B 0,C 180,E1 -9820.962,E2 -9820.962} C_VEL
LIN {X 0,Y 425.463,Z 432.42,A -85,B 0,C 180,E1 -9822.159,E2 -9822.159} C_VEL
LIN {X 0,Y 426.038,Z 422.518,A -85,B 0,C 180,E1 -9823.275,E2 -9823.275} C_VEL
LIN {X 0,Y 426.729,Z 411.178,A -85,B 0,C 180,E1 -9824.303,E2 -9824.303} C_VEL
LIN {X 0,Y 427.521,Z 399.543,A -85,B 0,C 180,E1 -9825.128,E2 -9825.128} C_VEL
LIN {X 0,Y 428.138,Z 387.451,A -85,B 0,C 180,E1 -9825.777,E2 -9825.777} C_VEL
LIN {X 0,Y 428.715,Z 374.393,A -85,B 0,C 180,E1 -9826.274,E2 -9826.274} C_VEL
LIN {X 0,Y 429.024,Z 360.342,A -85,B 0,C 180,E1 -9826.598,E2 -9826.598} C_VEL
LIN {X 0,Y 429.901,Z 285.545,A -85,B 0,C 180,E1 -9827.998,E2 -9827.998} C_VEL
LIN {X 0,Y 427.161,Z 262.472,A -85,B 0,C 180,E1 -9828.602,E2 -9828.602} C_VEL
LIN {X 0,Y 427.217,Z 259.642,A -85,B 0,C 180,E1 -9828.935,E2 -9828.935} C_VEL
LIN {X 0,Y 428.645,Z 233.471,A -85,B 0,C 180,E1 -9832.663,E2 -9832.663} C_VEL
LIN {X 0,Y 429.981,Z 212.241,A -85,B 0,C 180,E1 -9835.725,E2 -9835.725} C_VEL
LIN {X 0,Y 428.48,Z 203.994,A -85,B 0,C 180,E1 -9837.076,E2 -9837.076} C_VEL
LIN {X 0,Y 425.339,Z 191.683,A -85,B 0,C 180,E1 -9839.246,E2 -9839.246} C_VEL
LIN {X 0,Y 425.284,Z 191.512,A -85,B 0,C 180,E1 -9842.563,E2 -9842.563} C_VEL
LIN {X 0,Y 425.301,Z 191.51,A -85,B 0,C 180,E1 -9845.336,E2 -9845.336} C_VEL
LIN {X 0,Y 425.283,Z 191.513,A -85,B 0,C 180,E1 -9848.901,E2 -9848.901} C_VEL
LIN {X 0,Y 425.263,Z 191.513,A -85,B 0,C 180,E1 -9852.655,E2 -9852.655} C_VEL
LIN {X 0,Y 425.288,Z 191.51,A -85,B 0,C 180,E1 -9855.283,E2 -9855.283} C_VEL
LIN {X 0,Y 425.27,Z 191.511,A -85,B 0,C 180,E1 -9858.62,E2 -9858.62} C_VEL
LIN {X 0,Y 425.3,Z 191.509,A -85,B 0,C 180,E1 -9861.101,E2 -9861.101} C_VEL
LIN {X 0,Y 425.3,Z 191.507,A -85,B 0,C 180,E1 -9864.664,E2 -9864.664} C_VEL
LIN {X 0,Y 425.267,Z 191.511,A -85,B 0,C 180,E1 -9868.073,E2 -9868.073} C_VEL
LIN {X 0,Y 425.333,Z 191.503,A -85,B 0,C 180,E1 -9871.368,E2 -9871.368} C_VEL
LIN {X 0,Y 425.356,Z 191.499,A -85,B 0,C 180,E1 -9873.505,E2 -9873.505} C_VEL
LIN {X 0,Y 425.307,Z 191.508,A -85,B 0,C 180,E1 -9876.634,E2 -9876.634} C_VEL
LIN {X 0,Y 425.33,Z 191.507,A -85,B 0,C 180,E1 -9880.364,E2 -9880.364} C_VEL
LIN {X 0,Y 425.39,Z 191.496,A -85,B 0,C 180,E1 -9883.688,E2 -9883.688} C_VEL
LIN {X 0,Y 425.414,Z 191.492,A -85,B 0,C 180,E1 -9887.598,E2 -9887.598} C_VEL
LIN {X 0,Y 425.41,Z 191.494,A -85,B 0,C 180,E1 -9891.449,E2 -9891.449} C_VEL
LIN {X 0,Y 425.54,Z 191.481,A -85,B 0,C 180,E1 -9894.313,E2 -9894.313} C_VEL
LIN {X 0,Y 425.593,Z 191.662,A -85,B 0,C 180,E1 -9897.278,E2 -9897.278} C_VEL
LIN {X 0,Y 427.472,Z 200.379,A -85,B 0,C 180,E1 -9899.058,E2 -9899.058} C_VEL
LIN {X 0,Y 427.192,Z 215.678,A -85,B 0,C 180,E1 -9901.885,E2 -9901.885} C_VEL
LIN {X 0,Y 426.984,Z 229.168,A -85,B 0,C 180,E1 -9904.365,E2 -9904.365} C_VEL
LIN {X 0,Y 428.014,Z 234.078,A -85,B 0,C 180,E1 -9904.576,E2 -9904.576} C_VEL
LIN {X 0,Y 430.048,Z 244.79,A -85,B 0,C 180,E1 -9904.921,E2 -9904.921} C_VEL
LIN {X 0,Y 428.703,Z 312.294,A -85,B 0,C 180,E1 -9906.382,E2 -9906.382} C_VEL
LIN {X 0,Y 428.495,Z 324.417,A -85,B 0,C 180,E1 -9906.829,E2 -9906.829} C_VEL
LIN {X 0,Y 428.111,Z 335.503,A -85,B 0,C 180,E1 -9907.427,E2 -9907.427} C_VEL
LIN {X 0,Y 427.694,Z 345.548,A -85,B 0,C 180,E1 -9908.147,E2 -9908.147} C_VEL
LIN {X 0,Y 427.155,Z 356.56,A -85,B 0,C 180,E1 -9909.183,E2 -9909.183} C_VEL
LIN {X 0,Y 426.655,Z 365.015,A -85,B 0,C 180,E1 -9910.199,E2 -9910.199} C_VEL
LIN {X 0,Y 426.145,Z 373.09,A -85,B 0,C 180,E1 -9911.414,E2 -9911.414} C_VEL
LIN {X 0,Y 425.668,Z 380.508,A -85,B 0,C 180,E1 -9912.86,E2 -9912.86} C_VEL
LIN {X 0,Y 425.246,Z 386.228,A -85,B 0,C 180,E1 -9914.353,E2 -9914.353} C_VEL
LIN {X 0,Y 424.927,Z 390.32,A -85,B 0,C 180,E1 -9915.836,E2 -9915.836} C_VEL
LIN {X 0,Y 424.738,Z 393.013,A -85,B 0,C 180,E1 -9917.327,E2 -9917.327} C_VEL
LIN {X 0,Y 424.595,Z 394.073,A -85,B 0,C 180,E1 -9918.33,E2 -9918.33} C_VEL
LIN {X 0,Y 424.566,Z 394.576,A -85,B 0,C 180,E1 -9919.344,E2 -9919.344} C_VEL
LIN {X 0,Y 424.504,Z 394.483,A -85,B 0,C 180,E1 -9920.344,E2 -9920.344} C_VEL
LIN {X 0,Y 424.535,Z 393.057,A -85,B 0,C 180,E1 -9922.019,E2 -9922.019} C_VEL
LIN {X 0,Y 424.669,Z 390.662,A -85,B 0,C 180,E1 -9923.402,E2 -9923.402} C_VEL
LIN {X 0,Y 424.894,Z 386.549,A -85,B 0,C 180,E1 -9924.946,E2 -9924.946} C_VEL
LIN {X 0,Y 425.141,Z 380.689,A -85,B 0,C 180,E1 -9926.508,E2 -9926.508} C_VEL
LIN {X 0,Y 425.431,Z 374.205,A -85,B 0,C 180,E1 -9927.819,E2 -9927.819} C_VEL
LIN {X 0,Y 425.779,Z 366.943,A -85,B 0,C 180,E1 -9928.975,E2 -9928.975} C_VEL
LIN {X 0,Y 426.209,Z 358.493,A -85,B 0,C 180,E1 -9930.057,E2 -9930.057} C_VEL
LIN {X 0,Y 426.597,Z 348.629,A -85,B 0,C 180,E1 -9931.054,E2 -9931.054} C_VEL
LIN {X 0,Y 426.975,Z 339.542,A -85,B 0,C 180,E1 -9931.783,E2 -9931.783} C_VEL
LIN {X 0,Y 427.281,Z 328.701,A -85,B 0,C 180,E1 -9932.453,E2 -9932.453} C_VEL
LIN {X 0,Y 427.492,Z 317.516,A -85,B 0,C 180,E1 -9932.958,E2 -9932.958} C_VEL
LIN {X 0,Y 427.652,Z 305.186,A -85,B 0,C 180,E1 -9933.308,E2 -9933.308} C_VEL
LIN {X 0,Y 428.398,Z 242.407,A -85,B 0,C 180,E1 -9934.527,E2 -9934.527} C_VEL
LIN {X 0,Y 426.041,Z 228.069,A -85,B 0,C 180,E1 -9934.921,E2 -9934.921} C_VEL
LIN {X 0,Y 426.09,Z 224.072,A -85,B 0,C 180,E1 -9935.679,E2 -9935.679} C_VEL
LIN {X 0,Y 426.475,Z 209.213,A -85,B 0,C 180,E1 -9938.771,E2 -9938.771} C_VEL
LIN {X 0,Y 426.656,Z 198.995,A -85,B 0,C 180,E1 -9940.935,E2 -9940.935} C_VEL
LIN {X 0,Y 425.342,Z 191.599,A -85,B 0,C 180,E1 -9942.644,E2 -9942.644} C_VEL
LIN {X 0,Y 425.26,Z 191.515,A -85,B 0,C 180,E1 -9946.044,E2 -9946.044} C_VEL
LIN {X 0,Y 425.272,Z 191.507,A -85,B 0,C 180,E1 -9948.621,E2 -9948.621} C_VEL
LIN {X 0,Y 425.295,Z 191.505,A -85,B 0,C 180,E1 -9951.101,E2 -9951.101} C_VEL
LIN {X 0,Y 425.299,Z 191.504,A -85,B 0,C 180,E1 -9954.664,E2 -9954.664} C_VEL
LIN {X 0,Y 425.263,Z 191.51,A -85,B 0,C 180,E1 -9958.073,E2 -9958.073} C_VEL
LIN {X 0,Y 425.33,Z 191.505,A -85,B 0,C 180,E1 -9961.367,E2 -9961.367} C_VEL
LIN {X 0,Y 425.294,Z 191.504,A -85,B 0,C 180,E1 -9964.554,E2 -9964.554} C_VEL
LIN {X 0,Y 425.286,Z 191.51,A -85,B 0,C 180,E1 -9967.661,E2 -9967.661} C_VEL
LIN {X 0,Y 425.296,Z 191.506,A -85,B 0,C 180,E1 -9969.849,E2 -9969.849} C_VEL
LIN {X 0,Y 424.652,Z 191.586,A -85,B 0,C 180,E1 -9970.64,E2 -9970.64} C_VEL
LIN {X 0,Y 421.814,Z 191.939,A -85,B 0,C 180,E1 -9971.925,E2 -9971.925} C_VEL
LIN {X 0,Y 419.403,Z 192.241,A -85,B 0,C 180,E1 -9972.963,E2 -9972.963} C_VEL
LIN {X 0,Y 418.372,Z 192.37,A -85,B 0,C 180,E1 -9973.764,E2 -9973.764} C_VEL
LIN {X 0,Y 418.291,Z 192.377,A -85,B 0,C 180,E1 -9974.036,E2 -9974.036} C_VEL
LIN {X 0,Y 418.354,Z 192.375,A -85,B 0,C 180,E1 -9977.385,E2 -9977.385} C_VEL
LIN {X 0,Y 418.34,Z 192.371,A -85,B 0,C 180,E1 -9980.328,E2 -9980.328} C_VEL
LIN {X 0,Y 418.492,Z 192.358,A -85,B 0,C 180,E1 -9983.248,E2 -9983.248} C_VEL
LIN {X 0,Y 418.338,Z 192.378,A -85,B 0,C 180,E1 -9985.181,E2 -9985.181} C_VEL
LIN {X 0,Y 418.542,Z 192.345,A -85,B 0,C 180,E1 -9988.075,E2 -9988.075} C_VEL
LIN {X 0,Y 418.67,Z 192.329,A -85,B 0,C 180,E1 -9989.999,E2 -9989.999} C_VEL
LIN {X 0,Y 418.508,Z 192.355,A -85,B 0,C 180,E1 -9992.887,E2 -9992.887} C_VEL
LIN {X 0,Y 418.484,Z 192.357,A -85,B 0,C 180,E1 -9996.75,E2 -9996.75} C_VEL
LIN {X 0,Y 418.338,Z 192.371,A -85,B 0,C 180,E1 -9999.671,E2 -9999.671} C_VEL
LIN {X 0,Y 418.342,Z 192.376,A -85,B 0,C 180,E1 -10003,E2 -10003} C_VEL
LIN {X 0,Y 418.308,Z 192.381,A -85,B 0,C 180,E1 -10006.735,E2 -10006.735} C_VEL
LIN {X 0,Y 418.266,Z 192.38,A -85,B 0,C 180,E1 -10009.79,E2 -10009.79} C_VEL
LIN {X 0,Y 418.233,Z 192.391,A -85,B 0,C 180,E1 -10012.735,E2 -10012.735} C_VEL
LIN {X 0,Y 418.266,Z 192.38,A -85,B 0,C 180,E1 -10015.903,E2 -10015.903} C_VEL
LIN {X 0,Y 418.259,Z 192.382,A -85,B 0,C 180,E1 -10019.161,E2 -10019.161} C_VEL
LIN {X 0,Y 418.251,Z 192.386,A -85,B 0,C 180,E1 -10022.843,E2 -10022.843} C_VEL
LIN {X 0,Y 418.243,Z 192.387,A -85,B 0,C 180,E1 -10026.238,E2 -10026.238} C_VEL
LIN {X 0,Y 418.258,Z 192.381,A -85,B 0,C 180,E1 -10029.68,E2 -10029.68} C_VEL
LIN {X 0,Y 418.278,Z 192.385,A -85,B 0,C 180,E1 -10032.329,E2 -10032.329} C_VEL
LIN {X 0,Y 418.243,Z 192.383,A -85,B 0,C 180,E1 -10035.11,E2 -10035.11} C_VEL
LIN {X 0,Y 418.249,Z 192.383,A -85,B 0,C 180,E1 -10037.769,E2 -10037.769} C_VEL
LIN {X 0,Y 418.258,Z 192.384,A -85,B 0,C 180,E1 -10040.617,E2 -10040.617} C_VEL
LIN {X 0,Y 418.238,Z 192.387,A -85,B 0,C 180,E1 -10043.976,E2 -10043.976} C_VEL
LIN {X 0,Y 418.252,Z 192.382,A -85,B 0,C 180,E1 -10047.155,E2 -10047.155} C_VEL
LIN {X 0,Y 418.266,Z 192.38,A -85,B 0,C 180,E1 -10050.839,E2 -10050.839} C_VEL
LIN {X 0,Y 418.262,Z 192.388,A -85,B 0,C 180,E1 -10054.096,E2 -10054.096} C_VEL
LIN {X 0,Y 418.229,Z 192.385,A -85,B 0,C 180,E1 -10057.264,E2 -10057.264} C_VEL
LIN {X 0,Y 418.275,Z 192.382,A -85,B 0,C 180,E1 -10060.364,E2 -10060.364} C_VEL
LIN {X 0,Y 418.317,Z 192.375,A -85,B 0,C 180,E1 -10063.405,E2 -10063.405} C_VEL
LIN {X 0,Y 418.338,Z 192.371,A -85,B 0,C 180,E1 -10066.999,E2 -10066.999} C_VEL
LIN {X 0,Y 418.334,Z 192.373,A -85,B 0,C 180,E1 -10070.329,E2 -10070.329} C_VEL
LIN {X 0,Y 418.484,Z 192.354,A -85,B 0,C 180,E1 -10073.249,E2 -10073.249} C_VEL
LIN {X 0,Y 418.331,Z 192.373,A -85,B 0,C 180,E1 -10075.182,E2 -10075.182} C_VEL
LIN {X 0,Y 418.533,Z 192.35,A -85,B 0,C 180,E1 -10078.076,E2 -10078.076} C_VEL
LIN {X 0,Y 418.664,Z 192.334,A -85,B 0,C 180,E1 -10080,E2 -10080} C_VEL
LIN {X 0,Y 418.493,Z 192.352,A -85,B 0,C 180,E1 -10082.888,E2 -10082.888} C_VEL
LIN {X 0,Y 418.483,Z 192.353,A -85,B 0,C 180,E1 -10086.752,E2 -10086.752} C_VEL
LIN {X 0,Y 418.392,Z 192.364,A -85,B 0,C 180,E1 -10088.696,E2 -10088.696} C_VEL
LIN {X 0,Y 418.308,Z 192.38,A -85,B 0,C 180,E1 -10091.632,E2 -10091.632} C_VEL
LIN {X 0,Y 418.295,Z 192.376,A -85,B 0,C 180,E1 -10094.598,E2 -10094.598} C_VEL
LIN {X 0,Y 418.28,Z 192.383,A -85,B 0,C 180,E1 -10097.605,E2 -10097.605} C_VEL
LIN {X 0,Y 418.243,Z 192.383,A -85,B 0,C 180,E1 -10100.664,E2 -10100.664} C_VEL
LIN {X 0,Y 418.281,Z 192.38,A -85,B 0,C 180,E1 -10103.782,E2 -10103.782} C_VEL
LIN {X 0,Y 418.304,Z 192.38,A -85,B 0,C 180,E1 -10107.071,E2 -10107.071} C_VEL
LIN {X 0,Y 418.239,Z 192.383,A -85,B 0,C 180,E1 -10110.273,E2 -10110.273} C_VEL
LIN {X 0,Y 418.242,Z 192.385,A -85,B 0,C 180,E1 -10113.678,E2 -10113.678} C_VEL
LIN {X 0,Y 418.235,Z 192.389,A -85,B 0,C 180,E1 -10117.225,E2 -10117.225} C_VEL
LIN {X 0,Y 418.242,Z 192.384,A -85,B 0,C 180,E1 -10119.683,E2 -10119.683} C_VEL
LIN {X 0,Y 418.225,Z 192.386,A -85,B 0,C 180,E1 -10122.322,E2 -10122.322} C_VEL
LIN {X 0,Y 418.232,Z 192.39,A -85,B 0,C 180,E1 -10125.11,E2 -10125.11} C_VEL
LIN {X 0,Y 418.231,Z 192.384,A -85,B 0,C 180,E1 -10127.767,E2 -10127.767} C_VEL
LIN {X 0,Y 418.242,Z 192.387,A -85,B 0,C 180,E1 -10130.622,E2 -10130.622} C_VEL
LIN {X 0,Y 418.24,Z 192.383,A -85,B 0,C 180,E1 -10133.977,E2 -10133.977} C_VEL
LIN {X 0,Y 418.256,Z 192.388,A -85,B 0,C 180,E1 -10137.157,E2 -10137.157} C_VEL
LIN {X 0,Y 418.285,Z 192.555,A -85,B 0,C 180,E1 -10140.669,E2 -10140.669} C_VEL
LIN {X 0,Y 422.03,Z 208.975,A -85,B 0,C 180,E1 -10143.494,E2 -10143.494} C_VEL
LIN {X 0,Y 422.755,Z 212.637,A -85,B 0,C 180,E1 -10144.1,E2 -10144.1} C_VEL
LIN {X 0,Y 421.747,Z 229.751,A -85,B 0,C 180,E1 -10146.687,E2 -10146.687} C_VEL
LIN {X 0,Y 420.119,Z 254.98,A -85,B 0,C 180,E1 -10150.454,E2 -10150.454} C_VEL
LIN {X 0,Y 419.716,Z 263.536,A -85,B 0,C 180,E1 -10151.687,E2 -10151.687} C_VEL
LIN {X 0,Y 422.162,Z 287.645,A -85,B 0,C 180,E1 -10152.25,E2 -10152.25} C_VEL
LIN {X 0,Y 421.232,Z 371.297,A -85,B 0,C 180,E1 -10153.804,E2 -10153.804} C_VEL
LIN {X 0,Y 420.786,Z 383.923,A -85,B 0,C 180,E1 -10154.222,E2 -10154.222} C_VEL
LIN {X 0,Y 420.219,Z 396.784,A -85,B 0,C 180,E1 -10154.852,E2 -10154.852} C_VEL
LIN {X 0,Y 419.55,Z 409.313,A -85,B 0,C 180,E1 -10155.696,E2 -10155.696} C_VEL
LIN {X 0,Y 418.935,Z 420.399,A -85,B 0,C 180,E1 -10156.657,E2 -10156.657} C_VEL
LIN {X 0,Y 418.501,Z 429.492,A -85,B 0,C 180,E1 -10157.637,E2 -10157.637} C_VEL
LIN {X 0,Y 417.986,Z 438.715,A -85,B 0,C 180,E1 -10158.852,E2 -10158.852} C_VEL
LIN {X 0,Y 417.571,Z 447.683,A -85,B 0,C 180,E1 -10160.311,E2 -10160.311} C_VEL
LIN {X 0,Y 417.408,Z 454.799,A -85,B 0,C 180,E1 -10161.773,E2 -10161.773} C_VEL
LIN {X 0,Y 417.312,Z 460.443,A -85,B 0,C 180,E1 -10163.231,E2 -10163.231} C_VEL
LIN {X 0,Y 417.275,Z 464.82,A -85,B 0,C 180,E1 -10164.686,E2 -10164.686} C_VEL
LIN {X 0,Y 417.337,Z 468.063,A -85,B 0,C 180,E1 -10166.138,E2 -10166.138} C_VEL
LIN {X 0,Y 417.416,Z 469.654,A -85,B 0,C 180,E1 -10167.105,E2 -10167.105} C_VEL
LIN {X 0,Y 417.34,Z 470.769,A -85,B 0,C 180,E1 -10168.071,E2 -10168.071} C_VEL
LIN {X 0,Y 417.268,Z 471.428,A -85,B 0,C 180,E1 -10169.036,E2 -10169.036} C_VEL
LIN {X 0,Y 417.272,Z 471.684,A -85,B 0,C 180,E1 -10170.001,E2 -10170.001} C_VEL
LIN {X 0,Y 417.269,Z 471.522,A -85,B 0,C 180,E1 -10170.966,E2 -10170.966} C_VEL
LIN {X 0,Y 417.34,Z 470.899,A -85,B 0,C 180,E1 -10171.931,E2 -10171.931} C_VEL
LIN {X 0,Y 417.369,Z 469.854,A -85,B 0,C 180,E1 -10172.896,E2 -10172.896} C_VEL
LIN {X 0,Y 417.305,Z 468.382,A -85,B 0,C 180,E1 -10173.863,E2 -10173.863} C_VEL
